LIN {X 0,Y 559.92,Z 996.15,A -85,B 0,C 180,E1 26542.512,E2 26542.512} C_VEL
LIN {X 0,Y 559.973,Z 989.657,A -85,B 0,C 180,E1 26540.271,E2 26540.271} C_VEL
LIN {X 0,Y 560.061,Z 982.262,A -85,B 0,C 180,E1 26538.26,E2 26538.26} C_VEL
LIN {X 0,Y 560.202,Z 972.761,A -85,B 0,C 180,E1 26536.152,E2 26536.152} C_VEL
LIN {X 0,Y 560.424,Z 961.483,A -85,B 0,C 180,E1 26534.055,E2 26534.055} C_VEL
LIN {X 0,Y 560.742,Z 948.646,A -85,B 0,C 180,E1 26532.035,E2 26532.035} C_VEL
LIN {X 0,Y 561.138,Z 934.193,A -85,B 0,C 180,E1 26530.106,E2 26530.106} C_VEL
LIN {X 0,Y 561.602,Z 918.797,A -85,B 0,C 180,E1 26528.333,E2 26528.333} C_VEL
LIN {X 0,Y 562.148,Z 901.727,A -85,B 0,C 180,E1 26526.635,E2 26526.635} C_VEL
LIN {X 0,Y 562.75,Z 883.794,A -85,B 0,C 180,E1 26525.1,E2 26525.1} C_VEL
LIN {X 0,Y 563.386,Z 864.761,A -85,B 0,C 180,E1 26523.721,E2 26523.721} C_VEL
LIN {X 0,Y 563.999,Z 844.815,A -85,B 0,C 180,E1 26522.499,E2 26522.499} C_VEL
LIN {X 0,Y 564.598,Z 825.21,A -85,B 0,C 180,E1 26521.497,E2 26521.497} C_VEL
LIN {X 0,Y 565.108,Z 804.841,A -85,B 0,C 180,E1 26520.656,E2 26520.656} C_VEL
LIN {X 0,Y 565.556,Z 782.74,A -85,B 0,C 180,E1 26519.949,E2 26519.949} C_VEL
LIN {X 0,Y 565.946,Z 761.19,A -85,B 0,C 180,E1 26519.454,E2 26519.454} C_VEL
LIN {X 0,Y 567.275,Z 543.866,A -85,B 0,C 180,E1 26516.321,E2 26516.321} C_VEL
LIN {X 0,Y 567.582,Z 462.459,A -85,B 0,C 180,E1 26515.12,E2 26515.12} C_VEL
LIN {X 0,Y 566.314,Z 454.968,A -85,B 0,C 180,E1 26514.909,E2 26514.909} C_VEL
LIN {X 0,Y 567.237,Z 411.986,A -85,B 0,C 180,E1 26512.196,E2 26512.196} C_VEL
LIN {X 0,Y 560.35,Z 396.389,A -85,B 0,C 180,E1 26510.568,E2 26510.568} C_VEL
LIN {X 0,Y 560.276,Z 395.939,A -85,B 0,C 180,E1 26510.278,E2 26510.278} C_VEL
LIN {X 0,Y 560.249,Z 395.947,A -85,B 0,C 180,E1 26507.025,E2 26507.025} C_VEL
LIN {X 0,Y 560.265,Z 395.941,A -85,B 0,C 180,E1 26503.681,E2 26503.681} C_VEL
LIN {X 0,Y 560.282,Z 395.942,A -85,B 0,C 180,E1 26500.364,E2 26500.364} C_VEL
LIN {X 0,Y 560.232,Z 395.947,A -85,B 0,C 180,E1 26497.088,E2 26497.088} C_VEL
LIN {X 0,Y 560.281,Z 395.945,A -85,B 0,C 180,E1 26493.833,E2 26493.833} C_VEL
LIN {X 0,Y 560.225,Z 395.947,A -85,B 0,C 180,E1 26490.663,E2 26490.663} C_VEL
LIN {X 0,Y 560.25,Z 395.947,A -85,B 0,C 180,E1 26487.415,E2 26487.415} C_VEL
LIN {X 0,Y 560.221,Z 395.947,A -85,B 0,C 180,E1 26484.348,E2 26484.348} C_VEL
LIN {X 0,Y 560.218,Z 395.947,A -85,B 0,C 180,E1 26481.022,E2 26481.022} C_VEL
LIN {X 0,Y 560.23,Z 395.948,A -85,B 0,C 180,E1 26477.975,E2 26477.975} C_VEL
LIN {X 0,Y 560.197,Z 395.947,A -85,B 0,C 180,E1 26474.681,E2 26474.681} C_VEL
LIN {X 0,Y 560.264,Z 395.947,A -85,B 0,C 180,E1 26471.529,E2 26471.529} C_VEL
LIN {X 0,Y 560.202,Z 395.946,A -85,B 0,C 180,E1 26468.312,E2 26468.312} C_VEL
LIN {X 0,Y 560.271,Z 395.946,A -85,B 0,C 180,E1 26465.119,E2 26465.119} C_VEL
LIN {X 0,Y 560.22,Z 395.946,A -85,B 0,C 180,E1 26461.943,E2 26461.943} C_VEL
LIN {X 0,Y 560.239,Z 395.945,A -85,B 0,C 180,E1 26458.568,E2 26458.568} C_VEL
LIN {X 0,Y 560.261,Z 395.946,A -85,B 0,C 180,E1 26455.393,E2 26455.393} C_VEL
LIN {X 0,Y 560.232,Z 395.946,A -85,B 0,C 180,E1 26452.076,E2 26452.076} C_VEL
LIN {X 0,Y 560.282,Z 395.944,A -85,B 0,C 180,E1 26448.887,E2 26448.887} C_VEL
LIN {X 0,Y 560.242,Z 395.946,A -85,B 0,C 180,E1 26445.636,E2 26445.636} C_VEL
LIN {X 0,Y 560.276,Z 395.941,A -85,B 0,C 180,E1 26442.339,E2 26442.339} C_VEL
LIN {X 0,Y 560.281,Z 395.941,A -85,B 0,C 180,E1 26438.949,E2 26438.949} C_VEL
LIN {X 0,Y 560.282,Z 395.941,A -85,B 0,C 180,E1 26436.242,E2 26436.242} C_VEL
LIN {X 0,Y 559.287,Z 396.064,A -85,B 0,C 180,E1 26435.455,E2 26435.455} C_VEL
LIN {X 0,Y 552.871,Z 396.865,A -85,B 0,C 180,E1 26433.243,E2 26433.243} C_VEL
LIN {X 0,Y 552.334,Z 396.924,A -85,B 0,C 180,E1 26432.667,E2 26432.667} C_VEL
LIN {X 0,Y 552.397,Z 397.316,A -85,B 0,C 180,E1 26432.24,E2 26432.24} C_VEL
LIN {X 0,Y 557.962,Z 412.47,A -85,B 0,C 180,E1 26430.505,E2 26430.505} C_VEL
LIN {X 0,Y 556.968,Z 452.354,A -85,B 0,C 180,E1 26427.431,E2 26427.431} C_VEL
LIN {X 0,Y 558.756,Z 463.241,A -85,B 0,C 180,E1 26427.151,E2 26427.151} C_VEL
LIN {X 0,Y 557.243,Z 713.555,A -85,B 0,C 180,E1 26423.618,E2 26423.618} C_VEL
LIN {X 0,Y 556.883,Z 733.935,A -85,B 0,C 180,E1 26423.144,E2 26423.144} C_VEL
LIN {X 0,Y 556.454,Z 753.084,A -85,B 0,C 180,E1 26422.519,E2 26422.519} C_VEL
LIN {X 0,Y 555.948,Z 772.8,A -85,B 0,C 180,E1 26421.682,E2 26421.682} C_VEL
LIN {X 0,Y 555.374,Z 791.75,A -85,B 0,C 180,E1 26420.675,E2 26420.675} C_VEL
LIN {X 0,Y 554.778,Z 810.212,A -85,B 0,C 180,E1 26419.478,E2 26419.478} C_VEL
LIN {X 0,Y 554.188,Z 827.589,A -85,B 0,C 180,E1 26418.121,E2 26418.121} C_VEL
LIN {X 0,Y 553.652,Z 843.71,A -85,B 0,C 180,E1 26416.633,E2 26416.633} C_VEL
LIN {X 0,Y 553.171,Z 858.492,A -85,B 0,C 180,E1 26415.03,E2 26415.03} C_VEL
LIN {X 0,Y 552.755,Z 872.818,A -85,B 0,C 180,E1 26413.199,E2 26413.199} C_VEL
LIN {X 0,Y 552.434,Z 885.237,A -85,B 0,C 180,E1 26411.313,E2 26411.313} C_VEL
LIN {X 0,Y 552.217,Z 895.965,A -85,B 0,C 180,E1 26409.363,E2 26409.363} C_VEL
LIN {X 0,Y 552.063,Z 905.093,A -85,B 0,C 180,E1 26407.349,E2 26407.349} C_VEL
LIN {X 0,Y 551.978,Z 912.761,A -85,B 0,C 180,E1 26405.219,E2 26405.219} C_VEL
LIN {X 0,Y 551.935,Z 918.327,A -85,B 0,C 180,E1 26403.164,E2 26403.164} C_VEL
LIN {X 0,Y 551.919,Z 922.392,A -85,B 0,C 180,E1 26401.03,E2 26401.03} C_VEL
LIN {X 0,Y 551.912,Z 924.818,A -85,B 0,C 180,E1 26398.806,E2 26398.806} C_VEL
LIN {X 0,Y 551.907,Z 925.449,A -85,B 0,C 180,E1 26396.695,E2 26396.695} C_VEL
LIN {X 0,Y 551.911,Z 924.457,A -85,B 0,C 180,E1 26394.571,E2 26394.571} C_VEL
LIN {X 0,Y 551.92,Z 921.593,A -85,B 0,C 180,E1 26392.358,E2 26392.358} C_VEL
LIN {X 0,Y 551.941,Z 917.367,A -85,B 0,C 180,E1 26390.351,E2 26390.351} C_VEL
LIN {X 0,Y 551.986,Z 911.309,A -85,B 0,C 180,E1 26388.259,E2 26388.259} C_VEL
LIN {X 0,Y 552.079,Z 903.952,A -85,B 0,C 180,E1 26386.285,E2 26386.285} C_VEL
LIN {X 0,Y 552.246,Z 894.517,A -85,B 0,C 180,E1 26384.252,E2 26384.252} C_VEL
LIN {X 0,Y 552.488,Z 883.101,A -85,B 0,C 180,E1 26382.241,E2 26382.241} C_VEL
LIN {X 0,Y 552.812,Z 870.701,A -85,B 0,C 180,E1 26380.418,E2 26380.418} C_VEL
LIN {X 0,Y 553.208,Z 857.202,A -85,B 0,C 180,E1 26378.73,E2 26378.73} C_VEL
LIN {X 0,Y 553.725,Z 841.406,A -85,B 0,C 180,E1 26377.051,E2 26377.051} C_VEL
LIN {X 0,Y 554.291,Z 824.528,A -85,B 0,C 180,E1 26375.536,E2 26375.536} C_VEL
LIN {X 0,Y 554.899,Z 806.565,A -85,B 0,C 180,E1 26374.183,E2 26374.183} C_VEL
LIN {X 0,Y 555.465,Z 788.406,A -85,B 0,C 180,E1 26373.042,E2 26373.042} C_VEL
LIN {X 0,Y 556.058,Z 769.286,A -85,B 0,C 180,E1 26372.059,E2 26372.059} C_VEL
LIN {X 0,Y 556.56,Z 749.527,A -85,B 0,C 180,E1 26371.259,E2 26371.259} C_VEL
LIN {X 0,Y 556.952,Z 729.557,A -85,B 0,C 180,E1 26370.649,E2 26370.649} C_VEL
LIN {X 0,Y 557.27,Z 708.606,A -85,B 0,C 180,E1 26370.21,E2 26370.21} C_VEL
LIN {X 0,Y 558.763,Z 462.012,A -85,B 0,C 180,E1 26366.741,E2 26366.741} C_VEL
LIN {X 0,Y 556.95,Z 451.832,A -85,B 0,C 180,E1 26366.447,E2 26366.447} C_VEL
LIN {X 0,Y 557.925,Z 412.19,A -85,B 0,C 180,E1 26363.384,E2 26363.384} C_VEL
LIN {X 0,Y 552.374,Z 397.163,A -85,B 0,C 180,E1 26361.672,E2 26361.672} C_VEL
LIN {X 0,Y 552.316,Z 396.929,A -85,B 0,C 180,E1 26358.3,E2 26358.3} C_VEL
LIN {X 0,Y 552.335,Z 396.934,A -85,B 0,C 180,E1 26354.996,E2 26354.996} C_VEL
LIN {X 0,Y 552.327,Z 396.925,A -85,B 0,C 180,E1 26351.638,E2 26351.638} C_VEL
LIN {X 0,Y 552.329,Z 396.919,A -85,B 0,C 180,E1 26348.215,E2 26348.215} C_VEL
LIN {X 0,Y 552.332,Z 396.929,A -85,B 0,C 180,E1 26344.822,E2 26344.822} C_VEL
LIN {X 0,Y 552.32,Z 396.932,A -85,B 0,C 180,E1 26341.567,E2 26341.567} C_VEL
LIN {X 0,Y 552.338,Z 396.931,A -85,B 0,C 180,E1 26338.211,E2 26338.211} C_VEL
LIN {X 0,Y 552.337,Z 396.923,A -85,B 0,C 180,E1 26334.853,E2 26334.853} C_VEL
LIN {X 0,Y 552.323,Z 396.929,A -85,B 0,C 180,E1 26331.448,E2 26331.448} C_VEL
LIN {X 0,Y 552.331,Z 396.933,A -85,B 0,C 180,E1 26328.087,E2 26328.087} C_VEL
LIN {X 0,Y 552.328,Z 396.929,A -85,B 0,C 180,E1 26324.765,E2 26324.765} C_VEL
LIN {X 0,Y 552.336,Z 396.932,A -85,B 0,C 180,E1 26321.3,E2 26321.3} C_VEL
LIN {X 0,Y 552.332,Z 396.929,A -85,B 0,C 180,E1 26317.988,E2 26317.988} C_VEL
LIN {X 0,Y 552.322,Z 396.932,A -85,B 0,C 180,E1 26314.641,E2 26314.641} C_VEL
LIN {X 0,Y 552.334,Z 396.93,A -85,B 0,C 180,E1 26311.301,E2 26311.301} C_VEL
LIN {X 0,Y 552.34,Z 396.927,A -85,B 0,C 180,E1 26307.843,E2 26307.843} C_VEL
LIN {X 0,Y 552.325,Z 396.932,A -85,B 0,C 180,E1 26304.415,E2 26304.415} C_VEL
LIN {X 0,Y 552.327,Z 396.931,A -85,B 0,C 180,E1 26301.115,E2 26301.115} C_VEL
LIN {X 0,Y 552.337,Z 396.928,A -85,B 0,C 180,E1 26297.706,E2 26297.706} C_VEL
LIN {X 0,Y 552.332,Z 396.931,A -85,B 0,C 180,E1 26294.253,E2 26294.253} C_VEL
LIN {X 0,Y 552.327,Z 396.931,A -85,B 0,C 180,E1 26290.958,E2 26290.958} C_VEL
LIN {X 0,Y 552.329,Z 396.928,A -85,B 0,C 180,E1 26287.594,E2 26287.594} C_VEL
LIN {X 0,Y 552.334,Z 396.934,A -85,B 0,C 180,E1 26284.257,E2 26284.257} C_VEL
LIN {X 0,Y 552.333,Z 396.928,A -85,B 0,C 180,E1 26280.83,E2 26280.83} C_VEL
LIN {X 0,Y 552.328,Z 396.931,A -85,B 0,C 180,E1 26277.51,E2 26277.51} C_VEL
LIN {X 0,Y 552.322,Z 396.933,A -85,B 0,C 180,E1 26274.182,E2 26274.182} C_VEL
LIN {X 0,Y 552.337,Z 396.928,A -85,B 0,C 180,E1 26270.834,E2 26270.834} C_VEL
LIN {X 0,Y 552.336,Z 396.933,A -85,B 0,C 180,E1 26267.348,E2 26267.348} C_VEL
LIN {X 0,Y 552.321,Z 396.93,A -85,B 0,C 180,E1 26264.001,E2 26264.001} C_VEL
LIN {X 0,Y 552.332,Z 396.93,A -85,B 0,C 180,E1 26260.654,E2 26260.654} C_VEL
LIN {X 0,Y 552.332,Z 396.934,A -85,B 0,C 180,E1 26257.32,E2 26257.32} C_VEL
LIN {X 0,Y 552.329,Z 396.929,A -85,B 0,C 180,E1 26253.883,E2 26253.883} C_VEL
LIN {X 0,Y 552.333,Z 396.934,A -85,B 0,C 180,E1 26250.545,E2 26250.545} C_VEL
LIN {X 0,Y 552.319,Z 396.931,A -85,B 0,C 180,E1 26247.23,E2 26247.23} C_VEL
LIN {X 0,Y 552.339,Z 396.93,A -85,B 0,C 180,E1 26243.834,E2 26243.834} C_VEL
LIN {X 0,Y 552.341,Z 396.934,A -85,B 0,C 180,E1 26240.417,E2 26240.417} C_VEL
LIN {X 0,Y 552.319,Z 396.932,A -85,B 0,C 180,E1 26237.104,E2 26237.104} C_VEL
LIN {X 0,Y 552.335,Z 396.933,A -85,B 0,C 180,E1 26233.751,E2 26233.751} C_VEL
LIN {X 0,Y 552.329,Z 396.929,A -85,B 0,C 180,E1 26230.349,E2 26230.349} C_VEL
LIN {X 0,Y 552.41,Z 397.394,A -85,B 0,C 180,E1 26230.038,E2 26230.038} C_VEL
LIN {X 0,Y 560.517,Z 415.82,A -85,B 0,C 180,E1 26228.081,E2 26228.081} C_VEL
LIN {X 0,Y 559.592,Z 455.684,A -85,B 0,C 180,E1 26225.558,E2 26225.558} C_VEL
LIN {X 0,Y 561.185,Z 466.213,A -85,B 0,C 180,E1 26225.279,E2 26225.279} C_VEL
LIN {X 0,Y 559.613,Z 686.518,A -85,B 0,C 180,E1 26222.062,E2 26222.062} C_VEL
LIN {X 0,Y 559.04,Z 762.278,A -85,B 0,C 180,E1 26220.946,E2 26220.946} C_VEL
LIN {X 0,Y 558.58,Z 783.721,A -85,B 0,C 180,E1 26220.437,E2 26220.437} C_VEL
LIN {X 0,Y 558.051,Z 805.52,A -85,B 0,C 180,E1 26219.724,E2 26219.724} C_VEL
LIN {X 0,Y 557.441,Z 826.358,A -85,B 0,C 180,E1 26218.85,E2 26218.85} C_VEL
LIN {X 0,Y 556.742,Z 845.724,A -85,B 0,C 180,E1 26217.837,E2 26217.837} C_VEL
LIN {X 0,Y 555.983,Z 866.308,A -85,B 0,C 180,E1 26216.546,E2 26216.546} C_VEL
LIN {X 0,Y 555.241,Z 885.093,A -85,B 0,C 180,E1 26215.151,E2 26215.151} C_VEL
LIN {X 0,Y 554.548,Z 902.884,A -85,B 0,C 180,E1 26213.597,E2 26213.597} C_VEL
LIN {X 0,Y 553.91,Z 919.519,A -85,B 0,C 180,E1 26211.904,E2 26211.904} C_VEL
LIN {X 0,Y 553.324,Z 935.858,A -85,B 0,C 180,E1 26209.971,E2 26209.971} C_VEL
LIN {X 0,Y 552.863,Z 950.032,A -85,B 0,C 180,E1 26208.016,E2 26208.016} C_VEL
LIN {X 0,Y 552.505,Z 962.724,A -85,B 0,C 180,E1 26205.968,E2 26205.968} C_VEL
LIN {X 0,Y 552.256,Z 973.324,A -85,B 0,C 180,E1 26203.935,E2 26203.935} C_VEL
LIN {X 0,Y 552.08,Z 983.061,A -85,B 0,C 180,E1 26201.705,E2 26201.705} C_VEL
LIN {X 0,Y 551.98,Z 990.584,A -85,B 0,C 180,E1 26199.595,E2 26199.595} C_VEL
LIN {X 0,Y 551.925,Z 996.394,A -85,B 0,C 180,E1 26197.497,E2 26197.497} C_VEL
LIN {X 0,Y 551.905,Z 1000.982,A -85,B 0,C 180,E1 26195.303,E2 26195.303} C_VEL
LIN {X 0,Y 551.907,Z 1003.783,A -85,B 0,C 180,E1 26193.222,E2 26193.222} C_VEL
LIN {X 0,Y 551.903,Z 1005.306,A -85,B 0,C 180,E1 26190.936,E2 26190.936} C_VEL
LIN {X 0,Y 551.909,Z 1005.238,A -85,B 0,C 180,E1 26188.757,E2 26188.757} C_VEL
LIN {X 0,Y 551.914,Z 1003.545,A -85,B 0,C 180,E1 26186.559,E2 26186.559} C_VEL
LIN {X 0,Y 551.925,Z 1000.225,A -85,B 0,C 180,E1 26184.284,E2 26184.284} C_VEL
LIN {X 0,Y 551.946,Z 995.642,A -85,B 0,C 180,E1 26182.194,E2 26182.194} C_VEL
LIN {X 0,Y 552.003,Z 989.184,A -85,B 0,C 180,E1 26179.989,E2 26179.989} C_VEL
LIN {X 0,Y 552.117,Z 981.441,A -85,B 0,C 180,E1 26177.876,E2 26177.876} C_VEL
LIN {X 0,Y 552.296,Z 971.788,A -85,B 0,C 180,E1 26175.749,E2 26175.749} C_VEL
LIN {X 0,Y 552.579,Z 960.21,A -85,B 0,C 180,E1 26173.607,E2 26173.607} C_VEL
LIN {X 0,Y 552.936,Z 947.895,A -85,B 0,C 180,E1 26171.664,E2 26171.664} C_VEL
LIN {X 0,Y 553.409,Z 933.343,A -85,B 0,C 180,E1 26169.706,E2 26169.706} C_VEL
LIN {X 0,Y 553.971,Z 917.688,A -85,B 0,C 180,E1 26167.897,E2 26167.897} C_VEL
LIN {X 0,Y 554.661,Z 899.917,A -85,B 0,C 180,E1 26166.131,E2 26166.131} C_VEL
LIN {X 0,Y 555.379,Z 881.775,A -85,B 0,C 180,E1 26164.588,E2 26164.588} C_VEL
LIN {X 0,Y 556.106,Z 863.135,A -85,B 0,C 180,E1 26163.235,E2 26163.235} C_VEL
LIN {X 0,Y 556.812,Z 843.817,A -85,B 0,C 180,E1 26162.055,E2 26162.055} C_VEL
LIN {X 0,Y 557.492,Z 823.942,A -85,B 0,C 180,E1 26161.041,E2 26161.041} C_VEL
LIN {X 0,Y 558.103,Z 804.099,A -85,B 0,C 180,E1 26160.222,E2 26160.222} C_VEL
LIN {X 0,Y 558.603,Z 782.221,A -85,B 0,C 180,E1 26159.521,E2 26159.521} C_VEL
LIN {X 0,Y 559.058,Z 760.334,A -85,B 0,C 180,E1 26159.021,E2 26159.021} C_VEL
LIN {X 0,Y 560.682,Z 534.694,A -85,B 0,C 180,E1 26155.731,E2 26155.731} C_VEL
LIN {X 0,Y 561.012,Z 463.917,A -85,B 0,C 180,E1 26154.674,E2 26154.674} C_VEL
LIN {X 0,Y 559.495,Z 454.665,A -85,B 0,C 180,E1 26154.401,E2 26154.401} C_VEL
LIN {X 0,Y 560.46,Z 415.329,A -85,B 0,C 180,E1 26151.882,E2 26151.882} C_VEL
LIN {X 0,Y 552.396,Z 397.288,A -85,B 0,C 180,E1 26149.945,E2 26149.945} C_VEL
LIN {X 0,Y 552.312,Z 396.928,A -85,B 0,C 180,E1 26149.175,E2 26149.175} C_VEL
LIN {X 0,Y 552.333,Z 396.928,A -85,B 0,C 180,E1 26145.795,E2 26145.795} C_VEL
LIN {X 0,Y 552.338,Z 396.923,A -85,B 0,C 180,E1 26142.395,E2 26142.395} C_VEL
LIN {X 0,Y 552.298,Z 396.936,A -85,B 0,C 180,E1 26139.184,E2 26139.184} C_VEL
LIN {X 0,Y 552.344,Z 396.934,A -85,B 0,C 180,E1 26135.909,E2 26135.909} C_VEL
LIN {X 0,Y 552.293,Z 396.935,A -85,B 0,C 180,E1 26132.649,E2 26132.649} C_VEL
LIN {X 0,Y 552.296,Z 396.937,A -85,B 0,C 180,E1 26129.246,E2 26129.246} C_VEL
LIN {X 0,Y 552.31,Z 396.932,A -85,B 0,C 180,E1 26126.123,E2 26126.123} C_VEL
LIN {X 0,Y 552.274,Z 396.938,A -85,B 0,C 180,E1 26122.862,E2 26122.862} C_VEL
LIN {X 0,Y 552.332,Z 396.935,A -85,B 0,C 180,E1 26119.676,E2 26119.676} C_VEL
LIN {X 0,Y 552.258,Z 396.939,A -85,B 0,C 180,E1 26116.514,E2 26116.514} C_VEL
LIN {X 0,Y 552.316,Z 396.938,A -85,B 0,C 180,E1 26113.291,E2 26113.291} C_VEL
LIN {X 0,Y 552.263,Z 396.938,A -85,B 0,C 180,E1 26110.22,E2 26110.22} C_VEL
LIN {X 0,Y 552.306,Z 396.936,A -85,B 0,C 180,E1 26106.966,E2 26106.966} C_VEL
LIN {X 0,Y 552.286,Z 396.937,A -85,B 0,C 180,E1 26103.841,E2 26103.841} C_VEL
LIN {X 0,Y 552.286,Z 396.935,A -85,B 0,C 180,E1 26100.415,E2 26100.415} C_VEL
LIN {X 0,Y 552.341,Z 396.935,A -85,B 0,C 180,E1 26097.198,E2 26097.198} C_VEL
LIN {X 0,Y 552.289,Z 396.935,A -85,B 0,C 180,E1 26093.972,E2 26093.972} C_VEL
LIN {X 0,Y 552.34,Z 396.932,A -85,B 0,C 180,E1 26090.728,E2 26090.728} C_VEL
LIN {X 0,Y 552.313,Z 396.937,A -85,B 0,C 180,E1 26087.453,E2 26087.453} C_VEL
LIN {X 0,Y 552.311,Z 396.932,A -85,B 0,C 180,E1 26084.028,E2 26084.028} C_VEL
LIN {X 0,Y 552.34,Z 396.934,A -85,B 0,C 180,E1 26080.764,E2 26080.764} C_VEL
LIN {X 0,Y 552.315,Z 396.929,A -85,B 0,C 180,E1 26077.431,E2 26077.431} C_VEL
LIN {X 0,Y 552.336,Z 396.935,A -85,B 0,C 180,E1 26074.018,E2 26074.018} C_VEL
LIN {X 0,Y 552.334,Z 396.924,A -85,B 0,C 180,E1 26072.667,E2 26072.667} C_VEL
LIN {X 0,Y 552.297,Z 397.934,A -85,B 0,C 180,E1 26072.317,E2 26072.317} C_VEL
LIN {X 0,Y 552.136,Z 402.018,A -85,B 0,C 180,E1 26071.841,E2 26071.841} C_VEL
LIN {X 0,Y 550.706,Z 423.331,A -85,B 0,C 180,E1 26070.151,E2 26070.151} C_VEL
LIN {X 0,Y 549.819,Z 452.552,A -85,B 0,C 180,E1 26067.865,E2 26067.865} C_VEL
LIN {X 0,Y 551.832,Z 464.588,A -85,B 0,C 180,E1 26067.551,E2 26067.551} C_VEL
LIN {X 0,Y 550.09,Z 713.472,A -85,B 0,C 180,E1 26063.995,E2 26063.995} C_VEL
LIN {X 0,Y 549.677,Z 733.913,A -85,B 0,C 180,E1 26063.515,E2 26063.515} C_VEL
LIN {X 0,Y 549.192,Z 753.177,A -85,B 0,C 180,E1 26062.879,E2 26062.879} C_VEL
LIN {X 0,Y 548.586,Z 773.344,A -85,B 0,C 180,E1 26062.008,E2 26062.008} C_VEL
LIN {X 0,Y 547.917,Z 792.321,A -85,B 0,C 180,E1 26060.981,E2 26060.981} C_VEL
LIN {X 0,Y 547.231,Z 810.861,A -85,B 0,C 180,E1 26059.756,E2 26059.756} C_VEL
LIN {X 0,Y 546.528,Z 828.961,A -85,B 0,C 180,E1 26058.315,E2 26058.315} C_VEL
LIN {X 0,Y 545.887,Z 845.633,A -85,B 0,C 180,E1 26056.73,E2 26056.73} C_VEL
LIN {X 0,Y 545.325,Z 860.61,A -85,B 0,C 180,E1 26055.046,E2 26055.046} C_VEL
LIN {X 0,Y 544.86,Z 874.255,A -85,B 0,C 180,E1 26053.237,E2 26053.237} C_VEL
LIN {X 0,Y 544.498,Z 886.454,A -85,B 0,C 180,E1 26051.319,E2 26051.319} C_VEL
LIN {X 0,Y 544.24,Z 897.278,A -85,B 0,C 180,E1 26049.275,E2 26049.275} C_VEL
LIN {X 0,Y 544.067,Z 906.256,A -85,B 0,C 180,E1 26047.197,E2 26047.197} C_VEL
LIN {X 0,Y 543.981,Z 913.418,A -85,B 0,C 180,E1 26045.117,E2 26045.117} C_VEL
LIN {X 0,Y 543.937,Z 919.031,A -85,B 0,C 180,E1 26042.96,E2 26042.96} C_VEL
LIN {X 0,Y 543.922,Z 922.75,A -85,B 0,C 180,E1 26040.851,E2 26040.851} C_VEL
LIN {X 0,Y 543.907,Z 924.922,A -85,B 0,C 180,E1 26038.668,E2 26038.668} C_VEL
LIN {X 0,Y 543.903,Z 925.39,A -85,B 0,C 180,E1 26036.412,E2 26036.412} C_VEL
LIN {X 0,Y 543.912,Z 924.151,A -85,B 0,C 180,E1 26034.246,E2 26034.246} C_VEL
LIN {X 0,Y 543.923,Z 921.293,A -85,B 0,C 180,E1 26032.108,E2 26032.108} C_VEL
LIN {X 0,Y 543.943,Z 916.735,A -85,B 0,C 180,E1 26029.99,E2 26029.99} C_VEL
LIN {X 0,Y 543.999,Z 910.818,A -85,B 0,C 180,E1 26027.983,E2 26027.983} C_VEL
LIN {X 0,Y 544.12,Z 902.924,A -85,B 0,C 180,E1 26025.888,E2 26025.888} C_VEL
LIN {X 0,Y 544.322,Z 893.767,A -85,B 0,C 180,E1 26023.921,E2 26023.921} C_VEL
LIN {X 0,Y 544.625,Z 882.329,A -85,B 0,C 180,E1 26021.896,E2 26021.896} C_VEL
LIN {X 0,Y 545.005,Z 869.718,A -85,B 0,C 180,E1 26020.034,E2 26020.034} C_VEL
LIN {X 0,Y 545.478,Z 856.038,A -85,B 0,C 180,E1 26018.324,E2 26018.324} C_VEL
LIN {X 0,Y 546.039,Z 841.098,A -85,B 0,C 180,E1 26016.728,E2 26016.728} C_VEL
LIN {X 0,Y 546.707,Z 824.144,A -85,B 0,C 180,E1 26015.191,E2 26015.191} C_VEL
LIN {X 0,Y 547.416,Z 806.094,A -85,B 0,C 180,E1 26013.82,E2 26013.82} C_VEL
LIN {X 0,Y 548.082,Z 787.805,A -85,B 0,C 180,E1 26012.664,E2 26012.664} C_VEL
LIN {X 0,Y 548.747,Z 768.515,A -85,B 0,C 180,E1 26011.668,E2 26011.668} C_VEL
LIN {X 0,Y 549.339,Z 748.562,A -85,B 0,C 180,E1 26010.858,E2 26010.858} C_VEL
LIN {X 0,Y 549.8,Z 728.444,A -85,B 0,C 180,E1 26010.248,E2 26010.248} C_VEL
LIN {X 0,Y 550.127,Z 707.886,A -85,B 0,C 180,E1 26009.822,E2 26009.822} C_VEL
LIN {X 0,Y 551.842,Z 463.422,A -85,B 0,C 180,E1 26006.343,E2 26006.343} C_VEL
LIN {X 0,Y 549.793,Z 452.315,A -85,B 0,C 180,E1 26006.035,E2 26006.035} C_VEL
LIN {X 0,Y 550.947,Z 415.541,A -85,B 0,C 180,E1 26003.142,E2 26003.142} C_VEL
LIN {X 0,Y 545.067,Z 400.264,A -85,B 0,C 180,E1 26001.392,E2 26001.392} C_VEL
LIN {X 0,Y 544.423,Z 398.102,A -85,B 0,C 180,E1 26001.097,E2 26001.097} C_VEL
LIN {X 0,Y 544.395,Z 397.906,A -85,B 0,C 180,E1 25997.697,E2 25997.697} C_VEL
LIN {X 0,Y 544.383,Z 397.92,A -85,B 0,C 180,E1 25994.244,E2 25994.244} C_VEL
LIN {X 0,Y 544.394,Z 397.916,A -85,B 0,C 180,E1 25990.916,E2 25990.916} C_VEL
LIN {X 0,Y 544.384,Z 397.9,A -85,B 0,C 180,E1 25987.539,E2 25987.539} C_VEL
LIN {X 0,Y 544.393,Z 397.925,A -85,B 0,C 180,E1 25984.078,E2 25984.078} C_VEL
LIN {X 0,Y 544.395,Z 397.92,A -85,B 0,C 180,E1 25980.74,E2 25980.74} C_VEL
LIN {X 0,Y 544.381,Z 397.922,A -85,B 0,C 180,E1 25977.441,E2 25977.441} C_VEL
LIN {X 0,Y 544.401,Z 397.92,A -85,B 0,C 180,E1 25974.003,E2 25974.003} C_VEL
LIN {X 0,Y 544.4,Z 397.911,A -85,B 0,C 180,E1 25970.544,E2 25970.544} C_VEL
LIN {X 0,Y 544.383,Z 397.915,A -85,B 0,C 180,E1 25967.188,E2 25967.188} C_VEL
LIN {X 0,Y 544.394,Z 397.923,A -85,B 0,C 180,E1 25963.822,E2 25963.822} C_VEL
LIN {X 0,Y 544.405,Z 397.914,A -85,B 0,C 180,E1 25960.341,E2 25960.341} C_VEL
LIN {X 0,Y 544.385,Z 397.917,A -85,B 0,C 180,E1 25956.913,E2 25956.913} C_VEL
LIN {X 0,Y 544.39,Z 397.923,A -85,B 0,C 180,E1 25953.503,E2 25953.503} C_VEL
LIN {X 0,Y 544.402,Z 397.914,A -85,B 0,C 180,E1 25950.093,E2 25950.093} C_VEL
LIN {X 0,Y 544.389,Z 397.915,A -85,B 0,C 180,E1 25946.625,E2 25946.625} C_VEL
LIN {X 0,Y 544.389,Z 397.92,A -85,B 0,C 180,E1 25943.259,E2 25943.259} C_VEL
LIN {X 0,Y 544.393,Z 397.911,A -85,B 0,C 180,E1 25939.864,E2 25939.864} C_VEL
LIN {X 0,Y 544.398,Z 397.922,A -85,B 0,C 180,E1 25936.43,E2 25936.43} C_VEL
LIN {X 0,Y 544.388,Z 397.916,A -85,B 0,C 180,E1 25933.057,E2 25933.057} C_VEL
LIN {X 0,Y 544.388,Z 397.914,A -85,B 0,C 180,E1 25929.728,E2 25929.728} C_VEL
LIN {X 0,Y 544.397,Z 397.923,A -85,B 0,C 180,E1 25926.327,E2 25926.327} C_VEL
LIN {X 0,Y 544.39,Z 397.91,A -85,B 0,C 180,E1 25922.843,E2 25922.843} C_VEL
LIN {X 0,Y 544.389,Z 397.918,A -85,B 0,C 180,E1 25919.474,E2 25919.474} C_VEL
LIN {X 0,Y 544.389,Z 397.92,A -85,B 0,C 180,E1 25916.104,E2 25916.104} C_VEL
LIN {X 0,Y 544.396,Z 397.909,A -85,B 0,C 180,E1 25912.614,E2 25912.614} C_VEL
LIN {X 0,Y 544.392,Z 397.919,A -85,B 0,C 180,E1 25909.203,E2 25909.203} C_VEL
LIN {X 0,Y 544.385,Z 397.921,A -85,B 0,C 180,E1 25905.861,E2 25905.861} C_VEL
LIN {X 0,Y 544.399,Z 397.915,A -85,B 0,C 180,E1 25902.47,E2 25902.47} C_VEL
LIN {X 0,Y 544.398,Z 397.919,A -85,B 0,C 180,E1 25899.014,E2 25899.014} C_VEL
LIN {X 0,Y 544.38,Z 397.921,A -85,B 0,C 180,E1 25895.645,E2 25895.645} C_VEL
LIN {X 0,Y 544.398,Z 397.916,A -85,B 0,C 180,E1 25892.284,E2 25892.284} C_VEL
LIN {X 0,Y 544.402,Z 397.922,A -85,B 0,C 180,E1 25888.807,E2 25888.807} C_VEL
LIN {X 0,Y 544.381,Z 397.921,A -85,B 0,C 180,E1 25885.371,E2 25885.371} C_VEL
LIN {X 0,Y 544.396,Z 397.919,A -85,B 0,C 180,E1 25881.993,E2 25881.993} C_VEL
LIN {X 0,Y 544.395,Z 397.923,A -85,B 0,C 180,E1 25878.61,E2 25878.61} C_VEL
LIN {X 0,Y 544.381,Z 397.908,A -85,B 0,C 180,E1 25875.148,E2 25875.148} C_VEL
LIN {X 0,Y 544.391,Z 397.897,A -85,B 0,C 180,E1 25871.815,E2 25871.815} C_VEL
LIN {X 0,Y 544.413,Z 398.164,A -85,B 0,C 180,E1 25870.668,E2 25870.668} C_VEL
LIN {X 0,Y 545.523,Z 401.136,A -85,B 0,C 180,E1 25870.317,E2 25870.317} C_VEL
LIN {X 0,Y 553.767,Z 419.076,A -85,B 0,C 180,E1 25868.408,E2 25868.408} C_VEL
LIN {X 0,Y 552.808,Z 455.62,A -85,B 0,C 180,E1 25866.063,E2 25866.063} C_VEL
LIN {X 0,Y 554.641,Z 467.677,A -85,B 0,C 180,E1 25865.735,E2 25865.735} C_VEL
LIN {X 0,Y 552.823,Z 687.917,A -85,B 0,C 180,E1 25862.483,E2 25862.483} C_VEL
LIN {X 0,Y 552.175,Z 762.278,A -85,B 0,C 180,E1 25861.374,E2 25861.374} C_VEL
LIN {X 0,Y 551.643,Z 783.852,A -85,B 0,C 180,E1 25860.858,E2 25860.858} C_VEL
LIN {X 0,Y 551.021,Z 806.182,A -85,B 0,C 180,E1 25860.116,E2 25860.116} C_VEL
LIN {X 0,Y 550.334,Z 826.358,A -85,B 0,C 180,E1 25859.258,E2 25859.258} C_VEL
LIN {X 0,Y 549.541,Z 845.727,A -85,B 0,C 180,E1 25858.234,E2 25858.234} C_VEL
LIN {X 0,Y 548.658,Z 866.305,A -85,B 0,C 180,E1 25856.929,E2 25856.929} C_VEL
LIN {X 0,Y 547.805,Z 885.09,A -85,B 0,C 180,E1 25855.517,E2 25855.517} C_VEL
LIN {X 0,Y 547.005,Z 902.886,A -85,B 0,C 180,E1 25853.942,E2 25853.942} C_VEL
LIN {X 0,Y 546.266,Z 919.164,A -85,B 0,C 180,E1 25852.266,E2 25852.266} C_VEL
LIN {X 0,Y 545.603,Z 935.008,A -85,B 0,C 180,E1 25850.378,E2 25850.378} C_VEL
LIN {X 0,Y 545.097,Z 948.63,A -85,B 0,C 180,E1 25848.501,E2 25848.501} C_VEL
LIN {X 0,Y 544.663,Z 961.453,A -85,B 0,C 180,E1 25846.423,E2 25846.423} C_VEL
LIN {X 0,Y 544.341,Z 972.806,A -85,B 0,C 180,E1 25844.251,E2 25844.251} C_VEL
LIN {X 0,Y 544.136,Z 982.247,A -85,B 0,C 180,E1 25842.094,E2 25842.094} C_VEL
LIN {X 0,Y 544.009,Z 989.877,A -85,B 0,C 180,E1 25839.951,E2 25839.951} C_VEL
LIN {X 0,Y 543.942,Z 996.14,A -85,B 0,C 180,E1 25837.714,E2 25837.714} C_VEL
LIN {X 0,Y 543.916,Z 1000.821,A -85,B 0,C 180,E1 25835.487,E2 25835.487} C_VEL
LIN {X 0,Y 543.909,Z 1003.783,A -85,B 0,C 180,E1 25833.269,E2 25833.269} C_VEL
LIN {X 0,Y 543.905,Z 1005.306,A -85,B 0,C 180,E1 25830.95,E2 25830.95} C_VEL
LIN {X 0,Y 543.908,Z 1005.238,A -85,B 0,C 180,E1 25828.738,E2 25828.738} C_VEL
LIN {X 0,Y 543.913,Z 1003.562,A -85,B 0,C 180,E1 25826.524,E2 25826.524} C_VEL
LIN {X 0,Y 543.925,Z 1000.431,A -85,B 0,C 180,E1 25824.306,E2 25824.306} C_VEL
LIN {X 0,Y 543.95,Z 995.896,A -85,B 0,C 180,E1 25822.185,E2 25822.185} C_VEL
LIN {X 0,Y 544.03,Z 989.185,A -85,B 0,C 180,E1 25819.84,E2 25819.84} C_VEL
LIN {X 0,Y 544.161,Z 981.441,A -85,B 0,C 180,E1 25817.696,E2 25817.696} C_VEL
LIN {X 0,Y 544.375,Z 971.789,A -85,B 0,C 180,E1 25815.538,E2 25815.538} C_VEL
LIN {X 0,Y 544.705,Z 960.21,A -85,B 0,C 180,E1 25813.363,E2 25813.363} C_VEL
LIN {X 0,Y 545.123,Z 947.894,A -85,B 0,C 180,E1 25811.392,E2 25811.392} C_VEL
LIN {X 0,Y 545.672,Z 933.344,A -85,B 0,C 180,E1 25809.405,E2 25809.405} C_VEL
LIN {X 0,Y 546.303,Z 918.194,A -85,B 0,C 180,E1 25807.627,E2 25807.627} C_VEL
LIN {X 0,Y 547.106,Z 900.522,A -85,B 0,C 180,E1 25805.838,E2 25805.838} C_VEL
LIN {X 0,Y 547.914,Z 883.073,A -85,B 0,C 180,E1 25804.32,E2 25804.32} C_VEL
LIN {X 0,Y 548.728,Z 864.64,A -85,B 0,C 180,E1 25802.954,E2 25802.954} C_VEL
LIN {X 0,Y 549.583,Z 844.708,A -85,B 0,C 180,E1 25801.707,E2 25801.707} C_VEL
LIN {X 0,Y 550.381,Z 824.65,A -85,B 0,C 180,E1 25800.663,E2 25800.663} C_VEL
LIN {X 0,Y 551.074,Z 804.836,A -85,B 0,C 180,E1 25799.833,E2 25799.833} C_VEL
LIN {X 0,Y 551.669,Z 782.611,A -85,B 0,C 180,E1 25799.108,E2 25799.108} C_VEL
LIN {X 0,Y 552.189,Z 760.869,A -85,B 0,C 180,E1 25798.602,E2 25798.602} C_VEL
LIN {X 0,Y 554.048,Z 537.366,A -85,B 0,C 180,E1 25795.304,E2 25795.304} C_VEL
LIN {X 0,Y 554.457,Z 465.295,A -85,B 0,C 180,E1 25794.214,E2 25794.214} C_VEL
LIN {X 0,Y 552.721,Z 454.694,A -85,B 0,C 180,E1 25793.899,E2 25793.899} C_VEL
LIN {X 0,Y 553.768,Z 419.073,A -85,B 0,C 180,E1 25791.592,E2 25791.592} C_VEL
LIN {X 0,Y 546.834,Z 404.135,A -85,B 0,C 180,E1 25790.006,E2 25790.006} C_VEL
LIN {X 0,Y 544.412,Z 398.202,A -85,B 0,C 180,E1 25789.355,E2 25789.355} C_VEL
LIN {X 0,Y 544.37,Z 397.926,A -85,B 0,C 180,E1 25787.126,E2 25787.126} C_VEL
LIN {X 0,Y 544.396,Z 397.918,A -85,B 0,C 180,E1 25783.802,E2 25783.802} C_VEL
LIN {X 0,Y 544.399,Z 397.921,A -85,B 0,C 180,E1 25780.415,E2 25780.415} C_VEL
LIN {X 0,Y 544.354,Z 397.925,A -85,B 0,C 180,E1 25777.046,E2 25777.046} C_VEL
LIN {X 0,Y 544.402,Z 397.923,A -85,B 0,C 180,E1 25773.813,E2 25773.813} C_VEL
LIN {X 0,Y 544.355,Z 397.924,A -85,B 0,C 180,E1 25770.528,E2 25770.528} C_VEL
LIN {X 0,Y 544.346,Z 397.923,A -85,B 0,C 180,E1 25767.099,E2 25767.099} C_VEL
LIN {X 0,Y 544.381,Z 397.924,A -85,B 0,C 180,E1 25763.948,E2 25763.948} C_VEL
LIN {X 0,Y 544.329,Z 397.925,A -85,B 0,C 180,E1 25760.763,E2 25760.763} C_VEL
LIN {X 0,Y 544.391,Z 397.923,A -85,B 0,C 180,E1 25757.53,E2 25757.53} C_VEL
LIN {X 0,Y 544.317,Z 397.925,A -85,B 0,C 180,E1 25754.358,E2 25754.358} C_VEL
LIN {X 0,Y 544.354,Z 397.927,A -85,B 0,C 180,E1 25751.012,E2 25751.012} C_VEL
LIN {X 0,Y 544.342,Z 397.923,A -85,B 0,C 180,E1 25747.918,E2 25747.918} C_VEL
LIN {X 0,Y 544.34,Z 397.925,A -85,B 0,C 180,E1 25744.53,E2 25744.53} C_VEL
LIN {X 0,Y 544.403,Z 397.923,A -85,B 0,C 180,E1 25741.263,E2 25741.263} C_VEL
LIN {X 0,Y 544.345,Z 397.925,A -85,B 0,C 180,E1 25738,E2 25738} C_VEL
LIN {X 0,Y 544.382,Z 397.921,A -85,B 0,C 180,E1 25734.625,E2 25734.625} C_VEL
LIN {X 0,Y 544.387,Z 397.926,A -85,B 0,C 180,E1 25731.338,E2 25731.338} C_VEL
LIN {X 0,Y 544.362,Z 397.923,A -85,B 0,C 180,E1 25728.021,E2 25728.021} C_VEL
LIN {X 0,Y 544.404,Z 397.921,A -85,B 0,C 180,E1 25724.773,E2 25724.773} C_VEL
LIN {X 0,Y 544.38,Z 397.926,A -85,B 0,C 180,E1 25721.381,E2 25721.381} C_VEL
LIN {X 0,Y 544.38,Z 397.913,A -85,B 0,C 180,E1 25717.881,E2 25717.881} C_VEL
LIN {X 0,Y 544.396,Z 397.918,A -85,B 0,C 180,E1 25714.546,E2 25714.546} C_VEL
LIN {X 0,Y 544.44,Z 398.198,A -85,B 0,C 180,E1 25712.83,E2 25712.83} C_VEL
LIN {X 0,Y 551.013,Z 415.543,A -85,B 0,C 180,E1 25710.782,E2 25710.782} C_VEL
LIN {X 0,Y 550.706,Z 423.331,A -85,B 0,C 180,E1 25710.151,E2 25710.151} C_VEL
LIN {X 0,Y 549.667,Z 427.669,A -85,B 0,C 180,E1 25709.867,E2 25709.867} C_VEL
LIN {X 0,Y 543.829,Z 439.733,A -85,B 0,C 180,E1 25709.295,E2 25709.295} C_VEL
LIN {X 0,Y 543.008,Z 443.458,A -85,B 0,C 180,E1 25709.044,E2 25709.044} C_VEL
LIN {X 0,Y 542.791,Z 452.86,A -85,B 0,C 180,E1 25708.324,E2 25708.324} C_VEL
LIN {X 0,Y 544.936,Z 465.984,A -85,B 0,C 180,E1 25707.959,E2 25707.959} C_VEL
LIN {X 0,Y 542.961,Z 713.427,A -85,B 0,C 180,E1 25704.38,E2 25704.38} C_VEL
LIN {X 0,Y 542.496,Z 733.915,A -85,B 0,C 180,E1 25703.895,E2 25703.895} C_VEL
LIN {X 0,Y 541.95,Z 753.328,A -85,B 0,C 180,E1 25703.245,E2 25703.245} C_VEL
LIN {X 0,Y 541.269,Z 773.177,A -85,B 0,C 180,E1 25702.379,E2 25702.379} C_VEL
LIN {X 0,Y 540.53,Z 791.732,A -85,B 0,C 180,E1 25701.369,E2 25701.369} C_VEL
LIN {X 0,Y 539.765,Z 810.232,A -85,B 0,C 180,E1 25700.139,E2 25700.139} C_VEL
LIN {X 0,Y 538.966,Z 828.16,A -85,B 0,C 180,E1 25698.7,E2 25698.7} C_VEL
LIN {X 0,Y 538.232,Z 844.586,A -85,B 0,C 180,E1 25697.131,E2 25697.131} C_VEL
LIN {X 0,Y 537.593,Z 859.267,A -85,B 0,C 180,E1 25695.478,E2 25695.478} C_VEL
LIN {X 0,Y 537.061,Z 872.865,A -85,B 0,C 180,E1 25693.681,E2 25693.681} C_VEL
LIN {X 0,Y 536.62,Z 885.547,A -85,B 0,C 180,E1 25691.692,E2 25691.692} C_VEL
LIN {X 0,Y 536.315,Z 896.577,A -85,B 0,C 180,E1 25689.608,E2 25689.608} C_VEL
LIN {X 0,Y 536.112,Z 905.448,A -85,B 0,C 180,E1 25687.567,E2 25687.567} C_VEL
LIN {X 0,Y 536,Z 912.984,A -85,B 0,C 180,E1 25685.394,E2 25685.394} C_VEL
LIN {X 0,Y 535.941,Z 918.54,A -85,B 0,C 180,E1 25683.26,E2 25683.26} C_VEL
LIN {X 0,Y 535.919,Z 922.485,A -85,B 0,C 180,E1 25681.09,E2 25681.09} C_VEL
LIN {X 0,Y 535.915,Z 924.797,A -85,B 0,C 180,E1 25678.892,E2 25678.892} C_VEL
LIN {X 0,Y 535.909,Z 925.455,A -85,B 0,C 180,E1 25676.717,E2 25676.717} C_VEL
LIN {X 0,Y 535.912,Z 924.522,A -85,B 0,C 180,E1 25674.582,E2 25674.582} C_VEL
LIN {X 0,Y 535.921,Z 921.812,A -85,B 0,C 180,E1 25672.368,E2 25672.368} C_VEL
LIN {X 0,Y 535.949,Z 917.447,A -85,B 0,C 180,E1 25670.187,E2 25670.187} C_VEL
LIN {X 0,Y 536.011,Z 911.14,A -85,B 0,C 180,E1 25667.947,E2 25667.947} C_VEL
LIN {X 0,Y 536.141,Z 903.714,A -85,B 0,C 180,E1 25665.908,E2 25665.908} C_VEL
LIN {X 0,Y 536.382,Z 894.167,A -85,B 0,C 180,E1 25663.801,E2 25663.801} C_VEL
LIN {X 0,Y 536.732,Z 882.596,A -85,B 0,C 180,E1 25661.713,E2 25661.713} C_VEL
LIN {X 0,Y 537.195,Z 869.496,A -85,B 0,C 180,E1 25659.749,E2 25659.749} C_VEL
LIN {X 0,Y 537.784,Z 854.872,A -85,B 0,C 180,E1 25657.905,E2 25657.905} C_VEL
LIN {X 0,Y 538.431,Z 839.712,A -85,B 0,C 180,E1 25656.288,E2 25656.288} C_VEL
LIN {X 0,Y 539.166,Z 823.13,A -85,B 0,C 180,E1 25654.784,E2 25654.784} C_VEL
LIN {X 0,Y 539.982,Z 804.85,A -85,B 0,C 180,E1 25653.395,E2 25653.395} C_VEL
LIN {X 0,Y 540.761,Z 786.251,A -85,B 0,C 180,E1 25652.223,E2 25652.223} C_VEL
LIN {X 0,Y 541.473,Z 767.722,A -85,B 0,C 180,E1 25651.267,E2 25651.267} C_VEL
LIN {X 0,Y 542.147,Z 747.386,A -85,B 0,C 180,E1 25650.44,E2 25650.44} C_VEL
LIN {X 0,Y 542.697,Z 726.764,A -85,B 0,C 180,E1 25649.823,E2 25649.823} C_VEL
LIN {X 0,Y 543.03,Z 706.253,A -85,B 0,C 180,E1 25649.409,E2 25649.409} C_VEL
LIN {X 0,Y 544.948,Z 464.839,A -85,B 0,C 180,E1 25645.934,E2 25645.934} C_VEL
LIN {X 0,Y 542.685,Z 452.145,A -85,B 0,C 180,E1 25645.56,E2 25645.56} C_VEL
LIN {X 0,Y 543.91,Z 418.664,A -85,B 0,C 180,E1 25642.87,E2 25642.87} C_VEL
LIN {X 0,Y 537.414,Z 401.808,A -85,B 0,C 180,E1 25640.899,E2 25640.899} C_VEL
LIN {X 0,Y 536.473,Z 399.104,A -85,B 0,C 180,E1 25640.531,E2 25640.531} C_VEL
LIN {X 0,Y 536.454,Z 398.89,A -85,B 0,C 180,E1 25637.184,E2 25637.184} C_VEL
LIN {X 0,Y 536.44,Z 398.905,A -85,B 0,C 180,E1 25633.874,E2 25633.874} C_VEL
LIN {X 0,Y 536.46,Z 398.914,A -85,B 0,C 180,E1 25630.396,E2 25630.396} C_VEL
LIN {X 0,Y 536.455,Z 398.886,A -85,B 0,C 180,E1 25626.956,E2 25626.956} C_VEL
LIN {X 0,Y 536.444,Z 398.909,A -85,B 0,C 180,E1 25623.545,E2 25623.545} C_VEL
LIN {X 0,Y 536.463,Z 398.911,A -85,B 0,C 180,E1 25620.074,E2 25620.074} C_VEL
LIN {X 0,Y 536.457,Z 398.909,A -85,B 0,C 180,E1 25616.615,E2 25616.615} C_VEL
LIN {X 0,Y 536.445,Z 398.91,A -85,B 0,C 180,E1 25613.25,E2 25613.25} C_VEL
LIN {X 0,Y 536.46,Z 398.909,A -85,B 0,C 180,E1 25609.833,E2 25609.833} C_VEL
LIN {X 0,Y 536.458,Z 398.9,A -85,B 0,C 180,E1 25606.316,E2 25606.316} C_VEL
LIN {X 0,Y 536.446,Z 398.905,A -85,B 0,C 180,E1 25602.903,E2 25602.903} C_VEL
LIN {X 0,Y 536.465,Z 398.912,A -85,B 0,C 180,E1 25599.461,E2 25599.461} C_VEL
LIN {X 0,Y 536.454,Z 398.901,A -85,B 0,C 180,E1 25595.952,E2 25595.952} C_VEL
LIN {X 0,Y 536.446,Z 398.905,A -85,B 0,C 180,E1 25592.592,E2 25592.592} C_VEL
LIN {X 0,Y 536.456,Z 398.91,A -85,B 0,C 180,E1 25589.231,E2 25589.231} C_VEL
LIN {X 0,Y 536.459,Z 398.897,A -85,B 0,C 180,E1 25585.739,E2 25585.739} C_VEL
LIN {X 0,Y 536.449,Z 398.909,A -85,B 0,C 180,E1 25582.348,E2 25582.348} C_VEL
LIN {X 0,Y 536.449,Z 398.904,A -85,B 0,C 180,E1 25579.037,E2 25579.037} C_VEL
LIN {X 0,Y 536.462,Z 398.902,A -85,B 0,C 180,E1 25575.569,E2 25575.569} C_VEL
LIN {X 0,Y 536.455,Z 398.913,A -85,B 0,C 180,E1 25572.159,E2 25572.159} C_VEL
LIN {X 0,Y 536.448,Z 398.903,A -85,B 0,C 180,E1 25568.792,E2 25568.792} C_VEL
LIN {X 0,Y 536.453,Z 398.906,A -85,B 0,C 180,E1 25565.455,E2 25565.455} C_VEL
LIN {X 0,Y 536.46,Z 398.907,A -85,B 0,C 180,E1 25562.03,E2 25562.03} C_VEL
LIN {X 0,Y 536.449,Z 398.904,A -85,B 0,C 180,E1 25558.612,E2 25558.612} C_VEL
LIN {X 0,Y 536.452,Z 398.908,A -85,B 0,C 180,E1 25555.189,E2 25555.189} C_VEL
LIN {X 0,Y 536.46,Z 398.906,A -85,B 0,C 180,E1 25551.749,E2 25551.749} C_VEL
LIN {X 0,Y 536.448,Z 398.904,A -85,B 0,C 180,E1 25548.279,E2 25548.279} C_VEL
LIN {X 0,Y 536.453,Z 398.908,A -85,B 0,C 180,E1 25544.875,E2 25544.875} C_VEL
LIN {X 0,Y 536.458,Z 398.912,A -85,B 0,C 180,E1 25541.415,E2 25541.415} C_VEL
LIN {X 0,Y 536.45,Z 398.906,A -85,B 0,C 180,E1 25537.999,E2 25537.999} C_VEL
LIN {X 0,Y 536.454,Z 398.91,A -85,B 0,C 180,E1 25534.616,E2 25534.616} C_VEL
LIN {X 0,Y 536.447,Z 398.909,A -85,B 0,C 180,E1 25531.258,E2 25531.258} C_VEL
LIN {X 0,Y 536.456,Z 398.903,A -85,B 0,C 180,E1 25527.788,E2 25527.788} C_VEL
LIN {X 0,Y 536.457,Z 398.912,A -85,B 0,C 180,E1 25524.354,E2 25524.354} C_VEL
LIN {X 0,Y 536.445,Z 398.912,A -85,B 0,C 180,E1 25520.951,E2 25520.951} C_VEL
LIN {X 0,Y 536.46,Z 398.907,A -85,B 0,C 180,E1 25517.568,E2 25517.568} C_VEL
LIN {X 0,Y 536.46,Z 398.911,A -85,B 0,C 180,E1 25514.147,E2 25514.147} C_VEL
LIN {X 0,Y 536.489,Z 399.11,A -85,B 0,C 180,E1 25511.282,E2 25511.282} C_VEL
LIN {X 0,Y 537.761,Z 402.414,A -85,B 0,C 180,E1 25510.881,E2 25510.881} C_VEL
LIN {X 0,Y 547.1,Z 422.785,A -85,B 0,C 180,E1 25508.706,E2 25508.706} C_VEL
LIN {X 0,Y 546.079,Z 455.645,A -85,B 0,C 180,E1 25506.579,E2 25506.579} C_VEL
LIN {X 0,Y 548.134,Z 469.076,A -85,B 0,C 180,E1 25506.204,E2 25506.204} C_VEL
LIN {X 0,Y 546.065,Z 689.19,A -85,B 0,C 180,E1 25502.916,E2 25502.916} C_VEL
LIN {X 0,Y 545.336,Z 762.473,A -85,B 0,C 180,E1 25501.809,E2 25501.809} C_VEL
LIN {X 0,Y 544.739,Z 784.112,A -85,B 0,C 180,E1 25501.285,E2 25501.285} C_VEL
LIN {X 0,Y 544.046,Z 806.179,A -85,B 0,C 180,E1 25500.543,E2 25500.543} C_VEL
LIN {X 0,Y 543.259,Z 826.357,A -85,B 0,C 180,E1 25499.677,E2 25499.677} C_VEL
LIN {X 0,Y 542.367,Z 845.73,A -85,B 0,C 180,E1 25498.642,E2 25498.642} C_VEL
LIN {X 0,Y 541.361,Z 866.179,A -85,B 0,C 180,E1 25497.331,E2 25497.331} C_VEL
LIN {X 0,Y 540.407,Z 885.087,A -85,B 0,C 180,E1 25495.892,E2 25495.892} C_VEL
LIN {X 0,Y 539.482,Z 902.887,A -85,B 0,C 180,E1 25494.297,E2 25494.297} C_VEL
LIN {X 0,Y 538.63,Z 919.163,A -85,B 0,C 180,E1 25492.599,E2 25492.599} C_VEL
LIN {X 0,Y 537.869,Z 935.009,A -85,B 0,C 180,E1 25490.685,E2 25490.685} C_VEL
LIN {X 0,Y 537.262,Z 949.195,A -85,B 0,C 180,E1 25488.692,E2 25488.692} C_VEL
LIN {X 0,Y 536.792,Z 961.451,A -85,B 0,C 180,E1 25486.671,E2 25486.671} C_VEL
LIN {X 0,Y 536.421,Z 972.807,A -85,B 0,C 180,E1 25484.466,E2 25484.466} C_VEL
LIN {X 0,Y 536.18,Z 982.252,A -85,B 0,C 180,E1 25482.275,E2 25482.275} C_VEL
LIN {X 0,Y 536.035,Z 989.877,A -85,B 0,C 180,E1 25480.1,E2 25480.1} C_VEL
LIN {X 0,Y 535.956,Z 996.14,A -85,B 0,C 180,E1 25477.829,E2 25477.829} C_VEL
LIN {X 0,Y 535.922,Z 1000.82,A -85,B 0,C 180,E1 25475.569,E2 25475.569} C_VEL
LIN {X 0,Y 535.911,Z 1003.783,A -85,B 0,C 180,E1 25473.318,E2 25473.318} C_VEL
LIN {X 0,Y 535.905,Z 1005.305,A -85,B 0,C 180,E1 25470.964,E2 25470.964} C_VEL
LIN {X 0,Y 535.907,Z 1005.238,A -85,B 0,C 180,E1 25468.719,E2 25468.719} C_VEL
LIN {X 0,Y 535.912,Z 1003.562,A -85,B 0,C 180,E1 25466.473,E2 25466.473} C_VEL
LIN {X 0,Y 535.928,Z 1000.431,A -85,B 0,C 180,E1 25464.22,E2 25464.22} C_VEL
LIN {X 0,Y 535.962,Z 995.896,A -85,B 0,C 180,E1 25462.068,E2 25462.068} C_VEL
LIN {X 0,Y 536.054,Z 989.185,A -85,B 0,C 180,E1 25459.688,E2 25459.688} C_VEL
LIN {X 0,Y 536.207,Z 981.44,A -85,B 0,C 180,E1 25457.511,E2 25457.511} C_VEL
LIN {X 0,Y 536.457,Z 971.752,A -85,B 0,C 180,E1 25455.311,E2 25455.311} C_VEL
LIN {X 0,Y 536.835,Z 960.209,A -85,B 0,C 180,E1 25453.112,E2 25453.112} C_VEL
LIN {X 0,Y 537.318,Z 947.892,A -85,B 0,C 180,E1 25451.111,E2 25451.111} C_VEL
LIN {X 0,Y 537.956,Z 933.345,A -85,B 0,C 180,E1 25449.096,E2 25449.096} C_VEL
LIN {X 0,Y 538.675,Z 918.194,A -85,B 0,C 180,E1 25447.293,E2 25447.293} C_VEL
LIN {X 0,Y 539.592,Z 900.524,A -85,B 0,C 180,E1 25445.48,E2 25445.48} C_VEL
LIN {X 0,Y 540.51,Z 883.308,A -85,B 0,C 180,E1 25443.961,E2 25443.961} C_VEL
LIN {X 0,Y 541.433,Z 864.751,A -85,B 0,C 180,E1 25442.568,E2 25442.568} C_VEL
LIN {X 0,Y 542.402,Z 844.909,A -85,B 0,C 180,E1 25441.31,E2 25441.31} C_VEL
LIN {X 0,Y 543.297,Z 825.222,A -85,B 0,C 180,E1 25440.27,E2 25440.27} C_VEL
LIN {X 0,Y 544.071,Z 805.574,A -85,B 0,C 180,E1 25439.434,E2 25439.434} C_VEL
LIN {X 0,Y 544.766,Z 783.001,A -85,B 0,C 180,E1 25438.684,E2 25438.684} C_VEL
LIN {X 0,Y 545.351,Z 761.405,A -85,B 0,C 180,E1 25438.172,E2 25438.172} C_VEL
LIN {X 0,Y 547.071,Z 579.989,A -85,B 0,C 180,E1 25435.465,E2 25435.465} C_VEL
LIN {X 0,Y 547.958,Z 466.754,A -85,B 0,C 180,E1 25433.746,E2 25433.746} C_VEL
LIN {X 0,Y 545.992,Z 454.694,A -85,B 0,C 180,E1 25433.382,E2 25433.382} C_VEL
LIN {X 0,Y 547.1,Z 422.786,A -85,B 0,C 180,E1 25431.294,E2 25431.294} C_VEL
LIN {X 0,Y 536.527,Z 399.383,A -85,B 0,C 180,E1 25428.799,E2 25428.799} C_VEL
LIN {X 0,Y 536.462,Z 398.899,A -85,B 0,C 180,E1 25428.364,E2 25428.364} C_VEL
LIN {X 0,Y 536.429,Z 398.914,A -85,B 0,C 180,E1 25425.06,E2 25425.06} C_VEL
LIN {X 0,Y 536.447,Z 398.914,A -85,B 0,C 180,E1 25421.639,E2 25421.639} C_VEL
LIN {X 0,Y 536.464,Z 398.91,A -85,B 0,C 180,E1 25418.227,E2 25418.227} C_VEL
LIN {X 0,Y 536.413,Z 398.914,A -85,B 0,C 180,E1 25414.906,E2 25414.906} C_VEL
LIN {X 0,Y 536.45,Z 398.913,A -85,B 0,C 180,E1 25411.583,E2 25411.583} C_VEL
LIN {X 0,Y 536.418,Z 398.913,A -85,B 0,C 180,E1 25408.379,E2 25408.379} C_VEL
LIN {X 0,Y 536.404,Z 398.915,A -85,B 0,C 180,E1 25405.032,E2 25405.032} C_VEL
LIN {X 0,Y 536.458,Z 398.914,A -85,B 0,C 180,E1 25401.771,E2 25401.771} C_VEL
LIN {X 0,Y 536.385,Z 398.915,A -85,B 0,C 180,E1 25398.475,E2 25398.475} C_VEL
LIN {X 0,Y 536.411,Z 398.913,A -85,B 0,C 180,E1 25395.127,E2 25395.127} C_VEL
LIN {X 0,Y 536.392,Z 398.917,A -85,B 0,C 180,E1 25392.05,E2 25392.05} C_VEL
LIN {X 0,Y 536.392,Z 398.912,A -85,B 0,C 180,E1 25388.576,E2 25388.576} C_VEL
LIN {X 0,Y 536.448,Z 398.912,A -85,B 0,C 180,E1 25385.454,E2 25385.454} C_VEL
LIN {X 0,Y 536.399,Z 398.912,A -85,B 0,C 180,E1 25382.136,E2 25382.136} C_VEL
LIN {X 0,Y 536.448,Z 398.911,A -85,B 0,C 180,E1 25378.825,E2 25378.825} C_VEL
LIN {X 0,Y 536.433,Z 398.912,A -85,B 0,C 180,E1 25375.51,E2 25375.51} C_VEL
LIN {X 0,Y 536.419,Z 398.913,A -85,B 0,C 180,E1 25372.179,E2 25372.179} C_VEL
LIN {X 0,Y 536.466,Z 398.909,A -85,B 0,C 180,E1 25368.823,E2 25368.823} C_VEL
LIN {X 0,Y 536.437,Z 398.914,A -85,B 0,C 180,E1 25365.426,E2 25365.426} C_VEL
LIN {X 0,Y 536.436,Z 398.911,A -85,B 0,C 180,E1 25361.976,E2 25361.976} C_VEL
LIN {X 0,Y 536.459,Z 398.902,A -85,B 0,C 180,E1 25358.688,E2 25358.688} C_VEL
LIN {X 0,Y 536.443,Z 398.904,A -85,B 0,C 180,E1 25355.322,E2 25355.322} C_VEL
LIN {X 0,Y 536.481,Z 399.188,A -85,B 0,C 180,E1 25353.429,E2 25353.429} C_VEL
LIN {X 0,Y 543.307,Z 416.706,A -85,B 0,C 180,E1 25351.293,E2 25351.293} C_VEL
LIN {X 0,Y 544.048,Z 419.273,A -85,B 0,C 180,E1 25351.013,E2 25351.013} C_VEL
LIN {X 0,Y 543.008,Z 443.458,A -85,B 0,C 180,E1 25349.044,E2 25349.044} C_VEL
LIN {X 0,Y 542.408,Z 449.228,A -85,B 0,C 180,E1 25348.704,E2 25348.704} C_VEL
LIN {X 0,Y 541.115,Z 456.652,A -85,B 0,C 180,E1 25348.481,E2 25348.481} C_VEL
LIN {X 0,Y 538.606,Z 471.28,A -85,B 0,C 180,E1 25348.326,E2 25348.326} C_VEL
LIN {X 0,Y 538.146,Z 478.144,A -85,B 0,C 180,E1 25348.25,E2 25348.25} C_VEL
LIN {X 0,Y 536.024,Z 700.396,A -85,B 0,C 180,E1 25344.988,E2 25344.988} C_VEL
LIN {X 0,Y 535.65,Z 721.912,A -85,B 0,C 180,E1 25344.594,E2 25344.594} C_VEL
LIN {X 0,Y 535.087,Z 742.465,A -85,B 0,C 180,E1 25344.018,E2 25344.018} C_VEL
LIN {X 0,Y 534.408,Z 762.38,A -85,B 0,C 180,E1 25343.256,E2 25343.256} C_VEL
LIN {X 0,Y 533.647,Z 780.951,A -85,B 0,C 180,E1 25342.352,E2 25342.352} C_VEL
LIN {X 0,Y 532.773,Z 800.29,A -85,B 0,C 180,E1 25341.184,E2 25341.184} C_VEL
LIN {X 0,Y 531.877,Z 818.42,A -85,B 0,C 180,E1 25339.849,E2 25339.849} C_VEL
LIN {X 0,Y 531.014,Z 835.25,A -85,B 0,C 180,E1 25338.371,E2 25338.371} C_VEL
LIN {X 0,Y 530.259,Z 850.362,A -85,B 0,C 180,E1 25336.805,E2 25336.805} C_VEL
LIN {X 0,Y 529.558,Z 865.208,A -85,B 0,C 180,E1 25334.999,E2 25334.999} C_VEL
LIN {X 0,Y 528.994,Z 878.542,A -85,B 0,C 180,E1 25333.077,E2 25333.077} C_VEL
LIN {X 0,Y 528.572,Z 890.1,A -85,B 0,C 180,E1 25331.096,E2 25331.096} C_VEL
LIN {X 0,Y 528.275,Z 899.986,A -85,B 0,C 180,E1 25329.065,E2 25329.065} C_VEL
LIN {X 0,Y 528.077,Z 908.573,A -85,B 0,C 180,E1 25326.88,E2 25326.88} C_VEL
LIN {X 0,Y 527.976,Z 915.192,A -85,B 0,C 180,E1 25324.725,E2 25324.725} C_VEL
LIN {X 0,Y 527.923,Z 920.19,A -85,B 0,C 180,E1 25322.536,E2 25322.536} C_VEL
LIN {X 0,Y 527.903,Z 923.498,A -85,B 0,C 180,E1 25320.374,E2 25320.374} C_VEL
LIN {X 0,Y 527.902,Z 925.206,A -85,B 0,C 180,E1 25318.259,E2 25318.259} C_VEL
LIN {X 0,Y 527.91,Z 925.321,A -85,B 0,C 180,E1 25316.063,E2 25316.063} C_VEL
LIN {X 0,Y 527.905,Z 923.797,A -85,B 0,C 180,E1 25313.821,E2 25313.821} C_VEL
LIN {X 0,Y 527.916,Z 920.529,A -85,B 0,C 180,E1 25311.554,E2 25311.554} C_VEL
LIN {X 0,Y 527.963,Z 915.836,A -85,B 0,C 180,E1 25309.418,E2 25309.418} C_VEL
LIN {X 0,Y 528.063,Z 909.471,A -85,B 0,C 180,E1 25307.291,E2 25307.291} C_VEL
LIN {X 0,Y 528.228,Z 901.683,A -85,B 0,C 180,E1 25305.252,E2 25305.252} C_VEL
LIN {X 0,Y 528.513,Z 891.68,A -85,B 0,C 180,E1 25303.119,E2 25303.119} C_VEL
LIN {X 0,Y 528.929,Z 880.307,A -85,B 0,C 180,E1 25301.114,E2 25301.114} C_VEL
LIN {X 0,Y 529.463,Z 867.637,A -85,B 0,C 180,E1 25299.234,E2 25299.234} C_VEL
LIN {X 0,Y 530.116,Z 853.688,A -85,B 0,C 180,E1 25297.475,E2 25297.475} C_VEL
LIN {X 0,Y 530.903,Z 837.779,A -85,B 0,C 180,E1 25295.78,E2 25295.78} C_VEL
LIN {X 0,Y 531.749,Z 820.815,A -85,B 0,C 180,E1 25294.257,E2 25294.257} C_VEL
LIN {X 0,Y 532.59,Z 803.522,A -85,B 0,C 180,E1 25292.952,E2 25292.952} C_VEL
LIN {X 0,Y 533.471,Z 784.685,A -85,B 0,C 180,E1 25291.77,E2 25291.77} C_VEL
LIN {X 0,Y 534.278,Z 765.705,A -85,B 0,C 180,E1 25290.802,E2 25290.802} C_VEL
LIN {X 0,Y 534.973,Z 746.096,A -85,B 0,C 180,E1 25290.011,E2 25290.011} C_VEL
LIN {X 0,Y 535.605,Z 725.438,A -85,B 0,C 180,E1 25289.396,E2 25289.396} C_VEL
LIN {X 0,Y 535.977,Z 704.191,A -85,B 0,C 180,E1 25288.979,E2 25288.979} C_VEL
LIN {X 0,Y 538.212,Z 467.274,A -85,B 0,C 180,E1 25285.506,E2 25285.506} C_VEL
LIN {X 0,Y 535.714,Z 452.343,A -85,B 0,C 180,E1 25285.073,E2 25285.073} C_VEL
LIN {X 0,Y 536.965,Z 422.008,A -85,B 0,C 180,E1 25282.616,E2 25282.616} C_VEL
LIN {X 0,Y 530.652,Z 405.712,A -85,B 0,C 180,E1 25280.673,E2 25280.673} C_VEL
LIN {X 0,Y 528.539,Z 400.113,A -85,B 0,C 180,E1 25279.948,E2 25279.948} C_VEL
LIN {X 0,Y 528.511,Z 399.882,A -85,B 0,C 180,E1 25276.51,E2 25276.51} C_VEL
LIN {X 0,Y 528.517,Z 399.881,A -85,B 0,C 180,E1 25273.173,E2 25273.173} C_VEL
LIN {X 0,Y 528.504,Z 399.9,A -85,B 0,C 180,E1 25269.742,E2 25269.742} C_VEL
LIN {X 0,Y 528.517,Z 399.882,A -85,B 0,C 180,E1 25266.235,E2 25266.235} C_VEL
LIN {X 0,Y 528.517,Z 399.898,A -85,B 0,C 180,E1 25262.752,E2 25262.752} C_VEL
LIN {X 0,Y 528.505,Z 399.893,A -85,B 0,C 180,E1 25259.407,E2 25259.407} C_VEL
LIN {X 0,Y 528.519,Z 399.897,A -85,B 0,C 180,E1 25255.944,E2 25255.944} C_VEL
LIN {X 0,Y 528.517,Z 399.898,A -85,B 0,C 180,E1 25252.469,E2 25252.469} C_VEL
LIN {X 0,Y 528.506,Z 399.899,A -85,B 0,C 180,E1 25249.11,E2 25249.11} C_VEL
LIN {X 0,Y 528.522,Z 399.895,A -85,B 0,C 180,E1 25245.652,E2 25245.652} C_VEL
LIN {X 0,Y 528.515,Z 399.892,A -85,B 0,C 180,E1 25242.131,E2 25242.131} C_VEL
LIN {X 0,Y 528.507,Z 399.897,A -85,B 0,C 180,E1 25238.771,E2 25238.771} C_VEL
LIN {X 0,Y 528.518,Z 399.896,A -85,B 0,C 180,E1 25235.373,E2 25235.373} C_VEL
LIN {X 0,Y 528.518,Z 399.891,A -85,B 0,C 180,E1 25231.849,E2 25231.849} C_VEL
LIN {X 0,Y 528.508,Z 399.899,A -85,B 0,C 180,E1 25228.473,E2 25228.473} C_VEL
LIN {X 0,Y 528.518,Z 399.892,A -85,B 0,C 180,E1 25225.016,E2 25225.016} C_VEL
LIN {X 0,Y 528.518,Z 399.893,A -85,B 0,C 180,E1 25221.532,E2 25221.532} C_VEL
LIN {X 0,Y 528.511,Z 399.898,A -85,B 0,C 180,E1 25218.075,E2 25218.075} C_VEL
LIN {X 0,Y 528.518,Z 399.894,A -85,B 0,C 180,E1 25214.685,E2 25214.685} C_VEL
LIN {X 0,Y 528.515,Z 399.896,A -85,B 0,C 180,E1 25211.126,E2 25211.126} C_VEL
LIN {X 0,Y 528.511,Z 399.896,A -85,B 0,C 180,E1 25207.72,E2 25207.72} C_VEL
LIN {X 0,Y 528.515,Z 399.899,A -85,B 0,C 180,E1 25204.34,E2 25204.34} C_VEL
LIN {X 0,Y 528.518,Z 399.895,A -85,B 0,C 180,E1 25200.867,E2 25200.867} C_VEL
LIN {X 0,Y 528.512,Z 399.895,A -85,B 0,C 180,E1 25197.398,E2 25197.398} C_VEL
LIN {X 0,Y 528.517,Z 399.9,A -85,B 0,C 180,E1 25193.919,E2 25193.919} C_VEL
LIN {X 0,Y 528.514,Z 399.897,A -85,B 0,C 180,E1 25190.417,E2 25190.417} C_VEL
LIN {X 0,Y 528.515,Z 399.897,A -85,B 0,C 180,E1 25186.982,E2 25186.982} C_VEL
LIN {X 0,Y 528.515,Z 399.897,A -85,B 0,C 180,E1 25183.57,E2 25183.57} C_VEL
LIN {X 0,Y 528.514,Z 399.895,A -85,B 0,C 180,E1 25180.091,E2 25180.091} C_VEL
LIN {X 0,Y 528.516,Z 399.899,A -85,B 0,C 180,E1 25176.71,E2 25176.71} C_VEL
LIN {X 0,Y 528.512,Z 399.902,A -85,B 0,C 180,E1 25173.247,E2 25173.247} C_VEL
LIN {X 0,Y 528.515,Z 399.898,A -85,B 0,C 180,E1 25169.787,E2 25169.787} C_VEL
LIN {X 0,Y 528.517,Z 399.9,A -85,B 0,C 180,E1 25166.338,E2 25166.338} C_VEL
LIN {X 0,Y 528.506,Z 399.904,A -85,B 0,C 180,E1 25162.976,E2 25162.976} C_VEL
LIN {X 0,Y 528.52,Z 399.892,A -85,B 0,C 180,E1 25159.51,E2 25159.51} C_VEL
LIN {X 0,Y 528.514,Z 399.875,A -85,B 0,C 180,E1 25156.029,E2 25156.029} C_VEL
LIN {X 0,Y 528.501,Z 399.878,A -85,B 0,C 180,E1 25152.614,E2 25152.614} C_VEL
LIN {X 0,Y 528.556,Z 400.169,A -85,B 0,C 180,E1 25151.896,E2 25151.896} C_VEL
LIN {X 0,Y 531.186,Z 406.507,A -85,B 0,C 180,E1 25151.156,E2 25151.156} C_VEL
LIN {X 0,Y 540.314,Z 426.373,A -85,B 0,C 180,E1 25149.006,E2 25149.006} C_VEL
LIN {X 0,Y 539.4,Z 455.713,A -85,B 0,C 180,E1 25147.105,E2 25147.105} C_VEL
LIN {X 0,Y 541.663,Z 470.56,A -85,B 0,C 180,E1 25146.683,E2 25146.683} C_VEL
LIN {X 0,Y 539.336,Z 690.716,A -85,B 0,C 180,E1 25143.356,E2 25143.356} C_VEL
LIN {X 0,Y 538.534,Z 762.472,A -85,B 0,C 180,E1 25142.259,E2 25142.259} C_VEL
LIN {X 0,Y 537.872,Z 784.11,A -85,B 0,C 180,E1 25141.73,E2 25141.73} C_VEL
LIN {X 0,Y 537.101,Z 806.176,A -85,B 0,C 180,E1 25140.981,E2 25140.981} C_VEL
LIN {X 0,Y 536.202,Z 826.64,A -85,B 0,C 180,E1 25140.092,E2 25140.092} C_VEL
LIN {X 0,Y 535.179,Z 846.628,A -85,B 0,C 180,E1 25139.008,E2 25139.008} C_VEL
LIN {X 0,Y 534.04,Z 867.109,A -85,B 0,C 180,E1 25137.668,E2 25137.668} C_VEL
LIN {X 0,Y 532.98,Z 885.752,A -85,B 0,C 180,E1 25136.22,E2 25136.22} C_VEL
LIN {X 0,Y 531.963,Z 903.197,A -85,B 0,C 180,E1 25134.633,E2 25134.633} C_VEL
LIN {X 0,Y 530.988,Z 919.669,A -85,B 0,C 180,E1 25132.884,E2 25132.884} C_VEL
LIN {X 0,Y 530.109,Z 935.86,A -85,B 0,C 180,E1 25130.886,E2 25130.886} C_VEL
LIN {X 0,Y 529.418,Z 950.036,A -85,B 0,C 180,E1 25128.843,E2 25128.843} C_VEL
LIN {X 0,Y 528.877,Z 962.719,A -85,B 0,C 180,E1 25126.702,E2 25126.702} C_VEL
LIN {X 0,Y 528.485,Z 973.323,A -85,B 0,C 180,E1 25124.576,E2 25124.576} C_VEL
LIN {X 0,Y 528.197,Z 983.063,A -85,B 0,C 180,E1 25122.242,E2 25122.242} C_VEL
LIN {X 0,Y 528.039,Z 990.583,A -85,B 0,C 180,E1 25120.034,E2 25120.034} C_VEL
LIN {X 0,Y 527.951,Z 996.649,A -85,B 0,C 180,E1 25117.73,E2 25117.73} C_VEL
LIN {X 0,Y 527.908,Z 1001.3,A -85,B 0,C 180,E1 25115.327,E2 25115.327} C_VEL
LIN {X 0,Y 527.903,Z 1004.008,A -85,B 0,C 180,E1 25113.151,E2 25113.151} C_VEL
LIN {X 0,Y 527.896,Z 1005.35,A -85,B 0,C 180,E1 25110.762,E2 25110.762} C_VEL
LIN {X 0,Y 527.899,Z 1005.151,A -85,B 0,C 180,E1 25108.483,E2 25108.483} C_VEL
LIN {X 0,Y 527.909,Z 1003.336,A -85,B 0,C 180,E1 25106.202,E2 25106.202} C_VEL
LIN {X 0,Y 527.933,Z 999.814,A -85,B 0,C 180,E1 25103.805,E2 25103.805} C_VEL
LIN {X 0,Y 527.987,Z 994.878,A -85,B 0,C 180,E1 25101.508,E2 25101.508} C_VEL
LIN {X 0,Y 528.091,Z 988.121,A -85,B 0,C 180,E1 25099.199,E2 25099.199} C_VEL
LIN {X 0,Y 528.293,Z 979.609,A -85,B 0,C 180,E1 25096.876,E2 25096.876} C_VEL
LIN {X 0,Y 528.617,Z 969.7,A -85,B 0,C 180,E1 25094.648,E2 25094.648} C_VEL
LIN {X 0,Y 529.053,Z 958.29,A -85,B 0,C 180,E1 25092.516,E2 25092.516} C_VEL
LIN {X 0,Y 529.665,Z 944.809,A -85,B 0,C 180,E1 25090.369,E2 25090.369} C_VEL
LIN {X 0,Y 530.4,Z 930.678,A -85,B 0,C 180,E1 25088.436,E2 25088.436} C_VEL
LIN {X 0,Y 531.291,Z 914.839,A -85,B 0,C 180,E1 25086.571,E2 25086.571} C_VEL
LIN {X 0,Y 532.24,Z 898.092,A -85,B 0,C 180,E1 25084.881,E2 25084.881} C_VEL
LIN {X 0,Y 533.335,Z 879.439,A -85,B 0,C 180,E1 25083.264,E2 25083.264} C_VEL
LIN {X 0,Y 534.442,Z 860.595,A -85,B 0,C 180,E1 25081.875,E2 25081.875} C_VEL
LIN {X 0,Y 535.46,Z 840.894,A -85,B 0,C 180,E1 25080.658,E2 25080.658} C_VEL
LIN {X 0,Y 536.46,Z 821.02,A -85,B 0,C 180,E1 25079.648,E2 25079.648} C_VEL
LIN {X 0,Y 537.337,Z 800.476,A -85,B 0,C 180,E1 25078.798,E2 25078.798} C_VEL
LIN {X 0,Y 538.045,Z 779.484,A -85,B 0,C 180,E1 25078.142,E2 25078.142} C_VEL
LIN {X 0,Y 538.602,Z 757.084,A -85,B 0,C 180,E1 25077.646,E2 25077.646} C_VEL
LIN {X 0,Y 540.94,Z 536.857,A -85,B 0,C 180,E1 25074.329,E2 25074.329} C_VEL
LIN {X 0,Y 541.497,Z 468.241,A -85,B 0,C 180,E1 25073.267,E2 25073.267} C_VEL
LIN {X 0,Y 539.306,Z 454.896,A -85,B 0,C 180,E1 25072.864,E2 25072.864} C_VEL
LIN {X 0,Y 540.13,Z 425.748,A -85,B 0,C 180,E1 25070.946,E2 25070.946} C_VEL
LIN {X 0,Y 528.594,Z 400.356,A -85,B 0,C 180,E1 25068.182,E2 25068.182} C_VEL
LIN {X 0,Y 528.507,Z 399.899,A -85,B 0,C 180,E1 25067.667,E2 25067.667} C_VEL
LIN {X 0,Y 528.526,Z 399.902,A -85,B 0,C 180,E1 25064.199,E2 25064.199} C_VEL
LIN {X 0,Y 528.49,Z 399.902,A -85,B 0,C 180,E1 25060.826,E2 25060.826} C_VEL
LIN {X 0,Y 528.49,Z 399.905,A -85,B 0,C 180,E1 25057.388,E2 25057.388} C_VEL
LIN {X 0,Y 528.525,Z 399.899,A -85,B 0,C 180,E1 25054.051,E2 25054.051} C_VEL
LIN {X 0,Y 528.469,Z 399.904,A -85,B 0,C 180,E1 25050.719,E2 25050.719} C_VEL
LIN {X 0,Y 528.49,Z 399.901,A -85,B 0,C 180,E1 25047.37,E2 25047.37} C_VEL
LIN {X 0,Y 528.484,Z 399.903,A -85,B 0,C 180,E1 25044.12,E2 25044.12} C_VEL
LIN {X 0,Y 528.454,Z 399.902,A -85,B 0,C 180,E1 25040.836,E2 25040.836} C_VEL
LIN {X 0,Y 528.513,Z 399.9,A -85,B 0,C 180,E1 25037.558,E2 25037.558} C_VEL
LIN {X 0,Y 528.44,Z 399.902,A -85,B 0,C 180,E1 25034.351,E2 25034.351} C_VEL
LIN {X 0,Y 528.476,Z 399.905,A -85,B 0,C 180,E1 25031.016,E2 25031.016} C_VEL
LIN {X 0,Y 528.471,Z 399.901,A -85,B 0,C 180,E1 25027.829,E2 25027.829} C_VEL
LIN {X 0,Y 528.459,Z 399.903,A -85,B 0,C 180,E1 25024.42,E2 25024.42} C_VEL
LIN {X 0,Y 528.525,Z 399.902,A -85,B 0,C 180,E1 25021.084,E2 25021.084} C_VEL
LIN {X 0,Y 528.473,Z 399.904,A -85,B 0,C 180,E1 25017.831,E2 25017.831} C_VEL
LIN {X 0,Y 528.481,Z 399.901,A -85,B 0,C 180,E1 25014.321,E2 25014.321} C_VEL
LIN {X 0,Y 528.525,Z 399.899,A -85,B 0,C 180,E1 25011.076,E2 25011.076} C_VEL
LIN {X 0,Y 528.484,Z 399.902,A -85,B 0,C 180,E1 25007.766,E2 25007.766} C_VEL
LIN {X 0,Y 528.514,Z 399.898,A -85,B 0,C 180,E1 25004.338,E2 25004.338} C_VEL
LIN {X 0,Y 528.525,Z 399.9,A -85,B 0,C 180,E1 25000.896,E2 25000.896} C_VEL
LIN {X 0,Y 528.498,Z 399.892,A -85,B 0,C 180,E1 24997.532,E2 24997.532} C_VEL
LIN {X 0,Y 528.552,Z 400.122,A -85,B 0,C 180,E1 24994.063,E2 24994.063} C_VEL
LIN {X 0,Y 530.926,Z 406.275,A -85,B 0,C 180,E1 24993.25,E2 24993.25} C_VEL
LIN {X 0,Y 537.042,Z 421.871,A -85,B 0,C 180,E1 24991.353,E2 24991.353} C_VEL
LIN {X 0,Y 535.847,Z 452.765,A -85,B 0,C 180,E1 24988.838,E2 24988.838} C_VEL
LIN {X 0,Y 538.275,Z 467.291,A -85,B 0,C 180,E1 24988.415,E2 24988.415} C_VEL
LIN {X 0,Y 538.146,Z 478.144,A -85,B 0,C 180,E1 24988.25,E2 24988.25} C_VEL
LIN {X 0,Y 537.223,Z 485.84,A -85,B 0,C 180,E1 24988.195,E2 24988.195} C_VEL
LIN {X 0,Y 531.786,Z 506.374,A -85,B 0,C 180,E1 24988.263,E2 24988.263} C_VEL
LIN {X 0,Y 531.103,Z 512.976,A -85,B 0,C 180,E1 24988.208,E2 24988.208} C_VEL
LIN {X 0,Y 528.777,Z 714.373,A -85,B 0,C 180,E1 24985.165,E2 24985.165} C_VEL
LIN {X 0,Y 528.169,Z 736.078,A -85,B 0,C 180,E1 24984.624,E2 24984.624} C_VEL
LIN {X 0,Y 527.47,Z 755.297,A -85,B 0,C 180,E1 24983.944,E2 24983.944} C_VEL
LIN {X 0,Y 526.626,Z 774.677,A -85,B 0,C 180,E1 24983.058,E2 24983.058} C_VEL
LIN {X 0,Y 525.651,Z 794.155,A -85,B 0,C 180,E1 24981.945,E2 24981.945} C_VEL
LIN {X 0,Y 524.701,Z 812.283,A -85,B 0,C 180,E1 24980.678,E2 24980.678} C_VEL
LIN {X 0,Y 523.748,Z 829.506,A -85,B 0,C 180,E1 24979.239,E2 24979.239} C_VEL
LIN {X 0,Y 522.851,Z 845.463,A -85,B 0,C 180,E1 24977.659,E2 24977.659} C_VEL
LIN {X 0,Y 522.032,Z 860.436,A -85,B 0,C 180,E1 24975.905,E2 24975.905} C_VEL
LIN {X 0,Y 521.375,Z 873.441,A -85,B 0,C 180,E1 24974.113,E2 24974.113} C_VEL
LIN {X 0,Y 520.854,Z 885.345,A -85,B 0,C 180,E1 24972.184,E2 24972.184} C_VEL
LIN {X 0,Y 520.457,Z 895.996,A -85,B 0,C 180,E1 24970.128,E2 24970.128} C_VEL
LIN {X 0,Y 520.182,Z 905.096,A -85,B 0,C 180,E1 24967.994,E2 24967.994} C_VEL
LIN {X 0,Y 520.026,Z 912.658,A -85,B 0,C 180,E1 24965.764,E2 24965.764} C_VEL
LIN {X 0,Y 519.949,Z 918.452,A -85,B 0,C 180,E1 24963.493,E2 24963.493} C_VEL
LIN {X 0,Y 519.917,Z 922.399,A -85,B 0,C 180,E1 24961.277,E2 24961.277} C_VEL
LIN {X 0,Y 519.916,Z 924.796,A -85,B 0,C 180,E1 24958.952,E2 24958.952} C_VEL
LIN {X 0,Y 519.909,Z 925.461,A -85,B 0,C 180,E1 24956.741,E2 24956.741} C_VEL
LIN {X 0,Y 519.91,Z 924.454,A -85,B 0,C 180,E1 24954.42,E2 24954.42} C_VEL
LIN {X 0,Y 519.927,Z 921.686,A -85,B 0,C 180,E1 24952.14,E2 24952.14} C_VEL
LIN {X 0,Y 519.955,Z 917.528,A -85,B 0,C 180,E1 24950.013,E2 24950.013} C_VEL
LIN {X 0,Y 520.038,Z 911.553,A -85,B 0,C 180,E1 24947.797,E2 24947.797} C_VEL
LIN {X 0,Y 520.213,Z 904.052,A -85,B 0,C 180,E1 24945.648,E2 24945.648} C_VEL
LIN {X 0,Y 520.502,Z 894.928,A -85,B 0,C 180,E1 24943.551,E2 24943.551} C_VEL
LIN {X 0,Y 520.91,Z 884.141,A -85,B 0,C 180,E1 24941.512,E2 24941.512} C_VEL
LIN {X 0,Y 521.441,Z 872.106,A -85,B 0,C 180,E1 24939.6,E2 24939.6} C_VEL
LIN {X 0,Y 522.156,Z 857.968,A -85,B 0,C 180,E1 24937.701,E2 24937.701} C_VEL
LIN {X 0,Y 522.976,Z 842.843,A -85,B 0,C 180,E1 24935.978,E2 24935.978} C_VEL
LIN {X 0,Y 523.887,Z 826.837,A -85,B 0,C 180,E1 24934.431,E2 24934.431} C_VEL
LIN {X 0,Y 524.884,Z 809.272,A -85,B 0,C 180,E1 24933,E2 24933} C_VEL
LIN {X 0,Y 525.861,Z 790.626,A -85,B 0,C 180,E1 24931.741,E2 24931.741} C_VEL
LIN {X 0,Y 526.762,Z 771.795,A -85,B 0,C 180,E1 24930.705,E2 24930.705} C_VEL
LIN {X 0,Y 527.572,Z 752.626,A -85,B 0,C 180,E1 24929.862,E2 24929.862} C_VEL
LIN {X 0,Y 528.267,Z 732.081,A -85,B 0,C 180,E1 24929.174,E2 24929.174} C_VEL
LIN {X 0,Y 528.806,Z 711.691,A -85,B 0,C 180,E1 24928.698,E2 24928.698} C_VEL
LIN {X 0,Y 531.53,Z 467.466,A -85,B 0,C 180,E1 24925.027,E2 24925.027} C_VEL
LIN {X 0,Y 528.751,Z 452.088,A -85,B 0,C 180,E1 24924.545,E2 24924.545} C_VEL
LIN {X 0,Y 529.849,Z 424.866,A -85,B 0,C 180,E1 24922.298,E2 24922.298} C_VEL
LIN {X 0,Y 523.192,Z 407.682,A -85,B 0,C 180,E1 24920.205,E2 24920.205} C_VEL
LIN {X 0,Y 520.611,Z 401.105,A -85,B 0,C 180,E1 24919.331,E2 24919.331} C_VEL
LIN {X 0,Y 520.565,Z 400.879,A -85,B 0,C 180,E1 24915.993,E2 24915.993} C_VEL
LIN {X 0,Y 520.581,Z 400.864,A -85,B 0,C 180,E1 24912.563,E2 24912.563} C_VEL
LIN {X 0,Y 520.58,Z 400.887,A -85,B 0,C 180,E1 24909.067,E2 24909.067} C_VEL
LIN {X 0,Y 520.566,Z 400.885,A -85,B 0,C 180,E1 24905.608,E2 24905.608} C_VEL
LIN {X 0,Y 520.582,Z 400.887,A -85,B 0,C 180,E1 24902.068,E2 24902.068} C_VEL
LIN {X 0,Y 520.579,Z 400.881,A -85,B 0,C 180,E1 24898.633,E2 24898.633} C_VEL
LIN {X 0,Y 520.567,Z 400.88,A -85,B 0,C 180,E1 24895.217,E2 24895.217} C_VEL
LIN {X 0,Y 520.585,Z 400.884,A -85,B 0,C 180,E1 24891.771,E2 24891.771} C_VEL
LIN {X 0,Y 520.579,Z 400.886,A -85,B 0,C 180,E1 24888.344,E2 24888.344} C_VEL
LIN {X 0,Y 520.57,Z 400.886,A -85,B 0,C 180,E1 24884.866,E2 24884.866} C_VEL
LIN {X 0,Y 520.583,Z 400.883,A -85,B 0,C 180,E1 24881.324,E2 24881.324} C_VEL
LIN {X 0,Y 520.575,Z 400.886,A -85,B 0,C 180,E1 24877.869,E2 24877.869} C_VEL
LIN {X 0,Y 520.575,Z 400.886,A -85,B 0,C 180,E1 24874.38,E2 24874.38} C_VEL
LIN {X 0,Y 520.577,Z 400.883,A -85,B 0,C 180,E1 24870.845,E2 24870.845} C_VEL
LIN {X 0,Y 520.573,Z 400.887,A -85,B 0,C 180,E1 24867.45,E2 24867.45} C_VEL
LIN {X 0,Y 520.576,Z 400.884,A -85,B 0,C 180,E1 24864.028,E2 24864.028} C_VEL
LIN {X 0,Y 520.577,Z 400.879,A -85,B 0,C 180,E1 24860.461,E2 24860.461} C_VEL
LIN {X 0,Y 520.573,Z 400.889,A -85,B 0,C 180,E1 24856.959,E2 24856.959} C_VEL
LIN {X 0,Y 520.583,Z 400.879,A -85,B 0,C 180,E1 24853.439,E2 24853.439} C_VEL
LIN {X 0,Y 520.573,Z 400.882,A -85,B 0,C 180,E1 24849.955,E2 24849.955} C_VEL
LIN {X 0,Y 520.573,Z 400.887,A -85,B 0,C 180,E1 24846.507,E2 24846.507} C_VEL
LIN {X 0,Y 520.578,Z 400.873,A -85,B 0,C 180,E1 24842.973,E2 24842.973} C_VEL
LIN {X 0,Y 520.574,Z 400.885,A -85,B 0,C 180,E1 24839.56,E2 24839.56} C_VEL
LIN {X 0,Y 520.571,Z 400.886,A -85,B 0,C 180,E1 24836.146,E2 24836.146} C_VEL
LIN {X 0,Y 520.579,Z 400.874,A -85,B 0,C 180,E1 24832.607,E2 24832.607} C_VEL
LIN {X 0,Y 520.576,Z 400.884,A -85,B 0,C 180,E1 24829.151,E2 24829.151} C_VEL
LIN {X 0,Y 520.577,Z 400.89,A -85,B 0,C 180,E1 24825.655,E2 24825.655} C_VEL
LIN {X 0,Y 520.572,Z 400.884,A -85,B 0,C 180,E1 24822.103,E2 24822.103} C_VEL
LIN {X 0,Y 520.577,Z 400.885,A -85,B 0,C 180,E1 24818.676,E2 24818.676} C_VEL
LIN {X 0,Y 520.576,Z 400.885,A -85,B 0,C 180,E1 24815.247,E2 24815.247} C_VEL
LIN {X 0,Y 520.569,Z 400.884,A -85,B 0,C 180,E1 24811.679,E2 24811.679} C_VEL
LIN {X 0,Y 520.579,Z 400.882,A -85,B 0,C 180,E1 24808.247,E2 24808.247} C_VEL
LIN {X 0,Y 520.581,Z 400.886,A -85,B 0,C 180,E1 24804.716,E2 24804.716} C_VEL
LIN {X 0,Y 520.565,Z 400.888,A -85,B 0,C 180,E1 24801.233,E2 24801.233} C_VEL
LIN {X 0,Y 520.58,Z 400.887,A -85,B 0,C 180,E1 24797.85,E2 24797.85} C_VEL
LIN {X 0,Y 520.581,Z 400.882,A -85,B 0,C 180,E1 24794.358,E2 24794.358} C_VEL
LIN {X 0,Y 520.598,Z 401.105,A -85,B 0,C 180,E1 24792.572,E2 24792.572} C_VEL
LIN {X 0,Y 521.911,Z 404.378,A -85,B 0,C 180,E1 24792.15,E2 24792.15} C_VEL
LIN {X 0,Y 533.508,Z 429.679,A -85,B 0,C 180,E1 24789.323,E2 24789.323} C_VEL
LIN {X 0,Y 532.68,Z 455.609,A -85,B 0,C 180,E1 24787.641,E2 24787.641} C_VEL
LIN {X 0,Y 535.232,Z 471.976,A -85,B 0,C 180,E1 24787.174,E2 24787.174} C_VEL
LIN {X 0,Y 532.642,Z 692.116,A -85,B 0,C 180,E1 24783.809,E2 24783.809} C_VEL
LIN {X 0,Y 531.766,Z 762.472,A -85,B 0,C 180,E1 24782.72,E2 24782.72} C_VEL
LIN {X 0,Y 531.046,Z 784.107,A -85,B 0,C 180,E1 24782.187,E2 24782.187} C_VEL
LIN {X 0,Y 530.188,Z 806.173,A -85,B 0,C 180,E1 24781.43,E2 24781.43} C_VEL
LIN {X 0,Y 529.216,Z 826.354,A -85,B 0,C 180,E1 24780.547,E2 24780.547} C_VEL
LIN {X 0,Y 528.047,Z 846.852,A -85,B 0,C 180,E1 24779.424,E2 24779.424} C_VEL
LIN {X 0,Y 526.795,Z 867.105,A -85,B 0,C 180,E1 24778.082,E2 24778.082} C_VEL
LIN {X 0,Y 525.616,Z 885.788,A -85,B 0,C 180,E1 24776.612,E2 24776.612} C_VEL
LIN {X 0,Y 524.46,Z 903.494,A -85,B 0,C 180,E1 24774.98,E2 24774.98} C_VEL
LIN {X 0,Y 523.399,Z 919.626,A -85,B 0,C 180,E1 24773.24,E2 24773.24} C_VEL
LIN {X 0,Y 522.409,Z 935.858,A -85,B 0,C 180,E1 24771.209,E2 24771.209} C_VEL
LIN {X 0,Y 521.625,Z 950.038,A -85,B 0,C 180,E1 24769.136,E2 24769.136} C_VEL
LIN {X 0,Y 521.013,Z 962.718,A -85,B 0,C 180,E1 24766.962,E2 24766.962} C_VEL
LIN {X 0,Y 520.568,Z 973.322,A -85,B 0,C 180,E1 24764.802,E2 24764.802} C_VEL
LIN {X 0,Y 520.245,Z 983.064,A -85,B 0,C 180,E1 24762.432,E2 24762.432} C_VEL
LIN {X 0,Y 520.063,Z 990.71,A -85,B 0,C 180,E1 24760.149,E2 24760.149} C_VEL
LIN {X 0,Y 519.965,Z 996.649,A -85,B 0,C 180,E1 24757.849,E2 24757.849} C_VEL
LIN {X 0,Y 519.913,Z 1001.3,A -85,B 0,C 180,E1 24755.409,E2 24755.409} C_VEL
LIN {X 0,Y 519.905,Z 1004.008,A -85,B 0,C 180,E1 24753.199,E2 24753.199} C_VEL
LIN {X 0,Y 519.897,Z 1005.35,A -85,B 0,C 180,E1 24750.774,E2 24750.774} C_VEL
LIN {X 0,Y 519.899,Z 1005.151,A -85,B 0,C 180,E1 24748.46,E2 24748.46} C_VEL
LIN {X 0,Y 519.91,Z 1003.335,A -85,B 0,C 180,E1 24746.143,E2 24746.143} C_VEL
LIN {X 0,Y 519.938,Z 999.814,A -85,B 0,C 180,E1 24743.71,E2 24743.71} C_VEL
LIN {X 0,Y 519.993,Z 994.878,A -85,B 0,C 180,E1 24741.377,E2 24741.377} C_VEL
LIN {X 0,Y 520.115,Z 988.122,A -85,B 0,C 180,E1 24739.032,E2 24739.032} C_VEL
LIN {X 0,Y 520.348,Z 979.608,A -85,B 0,C 180,E1 24736.671,E2 24736.671} C_VEL
LIN {X 0,Y 520.717,Z 969.699,A -85,B 0,C 180,E1 24734.409,E2 24734.409} C_VEL
LIN {X 0,Y 521.212,Z 958.292,A -85,B 0,C 180,E1 24732.244,E2 24732.244} C_VEL
LIN {X 0,Y 521.903,Z 944.807,A -85,B 0,C 180,E1 24730.065,E2 24730.065} C_VEL
LIN {X 0,Y 522.734,Z 930.46,A -85,B 0,C 180,E1 24728.076,E2 24728.076} C_VEL
LIN {X 0,Y 523.739,Z 914.645,A -85,B 0,C 180,E1 24726.189,E2 24726.189} C_VEL
LIN {X 0,Y 524.831,Z 897.654,A -85,B 0,C 180,E1 24724.457,E2 24724.457} C_VEL
LIN {X 0,Y 526.042,Z 878.85,A -85,B 0,C 180,E1 24722.814,E2 24722.814} C_VEL
LIN {X 0,Y 527.293,Z 859.678,A -85,B 0,C 180,E1 24721.395,E2 24721.395} C_VEL
LIN {X 0,Y 528.383,Z 840.791,A -85,B 0,C 180,E1 24720.22,E2 24720.22} C_VEL
LIN {X 0,Y 529.521,Z 820.11,A -85,B 0,C 180,E1 24719.163,E2 24719.163} C_VEL
LIN {X 0,Y 530.485,Z 799.293,A -85,B 0,C 180,E1 24718.305,E2 24718.305} C_VEL
LIN {X 0,Y 531.263,Z 778.686,A -85,B 0,C 180,E1 24717.662,E2 24717.662} C_VEL
LIN {X 0,Y 531.853,Z 756.419,A -85,B 0,C 180,E1 24717.172,E2 24717.172} C_VEL
LIN {X 0,Y 534.437,Z 537.493,A -85,B 0,C 180,E1 24713.837,E2 24713.837} C_VEL
LIN {X 0,Y 535.071,Z 469.708,A -85,B 0,C 180,E1 24712.776,E2 24712.776} C_VEL
LIN {X 0,Y 532.579,Z 454.868,A -85,B 0,C 180,E1 24712.334,E2 24712.334} C_VEL
LIN {X 0,Y 533.425,Z 429.66,A -85,B 0,C 180,E1 24710.692,E2 24710.692} C_VEL
LIN {X 0,Y 521.722,Z 404.122,A -85,B 0,C 180,E1 24707.873,E2 24707.873} C_VEL
LIN {X 0,Y 520.592,Z 401.133,A -85,B 0,C 180,E1 24707.485,E2 24707.485} C_VEL
LIN {X 0,Y 520.588,Z 400.891,A -85,B 0,C 180,E1 24704.355,E2 24704.355} C_VEL
LIN {X 0,Y 520.548,Z 400.892,A -85,B 0,C 180,E1 24700.918,E2 24700.918} C_VEL
LIN {X 0,Y 520.559,Z 400.894,A -85,B 0,C 180,E1 24697.508,E2 24697.508} C_VEL
LIN {X 0,Y 520.583,Z 400.887,A -85,B 0,C 180,E1 24694.113,E2 24694.113} C_VEL
LIN {X 0,Y 520.529,Z 400.893,A -85,B 0,C 180,E1 24690.846,E2 24690.846} C_VEL
LIN {X 0,Y 520.561,Z 400.89,A -85,B 0,C 180,E1 24687.463,E2 24687.463} C_VEL
LIN {X 0,Y 520.541,Z 400.892,A -85,B 0,C 180,E1 24684.173,E2 24684.173} C_VEL
LIN {X 0,Y 520.515,Z 400.891,A -85,B 0,C 180,E1 24680.816,E2 24680.816} C_VEL
LIN {X 0,Y 520.574,Z 400.888,A -85,B 0,C 180,E1 24677.55,E2 24677.55} C_VEL
LIN {X 0,Y 520.505,Z 400.891,A -85,B 0,C 180,E1 24674.234,E2 24674.234} C_VEL
LIN {X 0,Y 520.516,Z 400.894,A -85,B 0,C 180,E1 24670.738,E2 24670.738} C_VEL
LIN {X 0,Y 520.579,Z 400.889,A -85,B 0,C 180,E1 24667.393,E2 24667.393} C_VEL
LIN {X 0,Y 520.521,Z 400.893,A -85,B 0,C 180,E1 24664.075,E2 24664.075} C_VEL
LIN {X 0,Y 520.546,Z 400.892,A -85,B 0,C 180,E1 24660.66,E2 24660.66} C_VEL
LIN {X 0,Y 520.572,Z 400.894,A -85,B 0,C 180,E1 24657.358,E2 24657.358} C_VEL
LIN {X 0,Y 520.536,Z 400.892,A -85,B 0,C 180,E1 24653.935,E2 24653.935} C_VEL
LIN {X 0,Y 520.567,Z 400.889,A -85,B 0,C 180,E1 24650.492,E2 24650.492} C_VEL
LIN {X 0,Y 520.581,Z 400.891,A -85,B 0,C 180,E1 24647.126,E2 24647.126} C_VEL
LIN {X 0,Y 520.551,Z 400.891,A -85,B 0,C 180,E1 24643.714,E2 24643.714} C_VEL
LIN {X 0,Y 520.579,Z 400.889,A -85,B 0,C 180,E1 24640.23,E2 24640.23} C_VEL
LIN {X 0,Y 520.585,Z 400.89,A -85,B 0,C 180,E1 24636.813,E2 24636.813} C_VEL
LIN {X 0,Y 520.613,Z 401.112,A -85,B 0,C 180,E1 24634.708,E2 24634.708} C_VEL
LIN {X 0,Y 528.579,Z 420.887,A -85,B 0,C 180,E1 24632.145,E2 24632.145} C_VEL
LIN {X 0,Y 530.186,Z 425.911,A -85,B 0,C 180,E1 24631.563,E2 24631.563} C_VEL
LIN {X 0,Y 528.965,Z 452.868,A -85,B 0,C 180,E1 24629.359,E2 24629.359} C_VEL
LIN {X 0,Y 531.679,Z 468.762,A -85,B 0,C 180,E1 24628.884,E2 24628.884} C_VEL
LIN {X 0,Y 531.103,Z 512.976,A -85,B 0,C 180,E1 24628.208,E2 24628.208} C_VEL
LIN {X 0,Y 530.2,Z 520.67,A -85,B 0,C 180,E1 24628.15,E2 24628.15} C_VEL
LIN {X 0,Y 524.729,Z 541.2,A -85,B 0,C 180,E1 24628.221,E2 24628.221} C_VEL
LIN {X 0,Y 524.024,Z 547.804,A -85,B 0,C 180,E1 24628.166,E2 24628.166} C_VEL
LIN {X 0,Y 521.884,Z 714.677,A -85,B 0,C 180,E1 24625.608,E2 24625.608} C_VEL
LIN {X 0,Y 521.223,Z 735.44,A -85,B 0,C 180,E1 24625.084,E2 24625.084} C_VEL
LIN {X 0,Y 520.438,Z 754.559,A -85,B 0,C 180,E1 24624.4,E2 24624.4} C_VEL
LIN {X 0,Y 519.451,Z 773.907,A -85,B 0,C 180,E1 24623.503,E2 24623.503} C_VEL
LIN {X 0,Y 518.36,Z 793.263,A -85,B 0,C 180,E1 24622.381,E2 24622.381} C_VEL
LIN {X 0,Y 517.35,Z 810.902,A -85,B 0,C 180,E1 24621.15,E2 24621.15} C_VEL
LIN {X 0,Y 516.27,Z 828.322,A -85,B 0,C 180,E1 24619.695,E2 24619.695} C_VEL
LIN {X 0,Y 515.256,Z 844.401,A -85,B 0,C 180,E1 24618.093,E2 24618.093} C_VEL
LIN {X 0,Y 514.369,Z 859.133,A -85,B 0,C 180,E1 24616.364,E2 24616.364} C_VEL
LIN {X 0,Y 513.603,Z 872.73,A -85,B 0,C 180,E1 24614.489,E2 24614.489} C_VEL
LIN {X 0,Y 512.972,Z 885.457,A -85,B 0,C 180,E1 24612.403,E2 24612.403} C_VEL
LIN {X 0,Y 512.523,Z 896.204,A -85,B 0,C 180,E1 24610.289,E2 24610.289} C_VEL
LIN {X 0,Y 512.215,Z 905.25,A -85,B 0,C 180,E1 24608.124,E2 24608.124} C_VEL
LIN {X 0,Y 512.039,Z 912.8,A -85,B 0,C 180,E1 24605.856,E2 24605.856} C_VEL
LIN {X 0,Y 511.955,Z 918.257,A -85,B 0,C 180,E1 24603.683,E2 24603.683} C_VEL
LIN {X 0,Y 511.918,Z 922.318,A -85,B 0,C 180,E1 24601.402,E2 24601.402} C_VEL
LIN {X 0,Y 511.911,Z 924.726,A -85,B 0,C 180,E1 24599.097,E2 24599.097} C_VEL
LIN {X 0,Y 511.912,Z 925.476,A -85,B 0,C 180,E1 24596.816,E2 24596.816} C_VEL
LIN {X 0,Y 511.912,Z 924.587,A -85,B 0,C 180,E1 24594.581,E2 24594.581} C_VEL
LIN {X 0,Y 511.923,Z 922.14,A -85,B 0,C 180,E1 24592.384,E2 24592.384} C_VEL
LIN {X 0,Y 511.959,Z 917.854,A -85,B 0,C 180,E1 24590.049,E2 24590.049} C_VEL
LIN {X 0,Y 512.046,Z 912.165,A -85,B 0,C 180,E1 24587.85,E2 24587.85} C_VEL
LIN {X 0,Y 512.239,Z 904.664,A -85,B 0,C 180,E1 24585.624,E2 24585.624} C_VEL
LIN {X 0,Y 512.562,Z 895.293,A -85,B 0,C 180,E1 24583.42,E2 24583.42} C_VEL
LIN {X 0,Y 513.016,Z 884.589,A -85,B 0,C 180,E1 24581.35,E2 24581.35} C_VEL
LIN {X 0,Y 513.607,Z 872.645,A -85,B 0,C 180,E1 24579.409,E2 24579.409} C_VEL
LIN {X 0,Y 514.397,Z 858.611,A -85,B 0,C 180,E1 24577.48,E2 24577.48} C_VEL
LIN {X 0,Y 515.304,Z 843.602,A -85,B 0,C 180,E1 24575.732,E2 24575.732} C_VEL
LIN {X 0,Y 516.297,Z 827.821,A -85,B 0,C 180,E1 24574.17,E2 24574.17} C_VEL
LIN {X 0,Y 517.39,Z 810.282,A -85,B 0,C 180,E1 24572.711,E2 24572.711} C_VEL
LIN {X 0,Y 518.456,Z 791.79,A -85,B 0,C 180,E1 24571.434,E2 24571.434} C_VEL
LIN {X 0,Y 519.531,Z 772.342,A -85,B 0,C 180,E1 24570.328,E2 24570.328} C_VEL
LIN {X 0,Y 520.488,Z 752.855,A -85,B 0,C 180,E1 24569.447,E2 24569.447} C_VEL
LIN {X 0,Y 521.284,Z 732.42,A -85,B 0,C 180,E1 24568.748,E2 24568.748} C_VEL
LIN {X 0,Y 521.878,Z 712.002,A -85,B 0,C 180,E1 24568.262,E2 24568.262} C_VEL
LIN {X 0,Y 524.916,Z 468.992,A -85,B 0,C 180,E1 24564.56,E2 24564.56} C_VEL
LIN {X 0,Y 521.844,Z 451.876,A -85,B 0,C 180,E1 24564.004,E2 24564.004} C_VEL
LIN {X 0,Y 522.964,Z 428.339,A -85,B 0,C 180,E1 24562.044,E2 24562.044} C_VEL
LIN {X 0,Y 516.448,Z 411.592,A -85,B 0,C 180,E1 24559.963,E2 24559.963} C_VEL
LIN {X 0,Y 512.668,Z 402.085,A -85,B 0,C 180,E1 24558.691,E2 24558.691} C_VEL
LIN {X 0,Y 512.645,Z 401.877,A -85,B 0,C 180,E1 24555.31,E2 24555.31} C_VEL
LIN {X 0,Y 512.626,Z 401.86,A -85,B 0,C 180,E1 24551.814,E2 24551.814} C_VEL
LIN {X 0,Y 512.644,Z 401.855,A -85,B 0,C 180,E1 24548.367,E2 24548.367} C_VEL
LIN {X 0,Y 512.64,Z 401.874,A -85,B 0,C 180,E1 24544.823,E2 24544.823} C_VEL
LIN {X 0,Y 512.634,Z 401.876,A -85,B 0,C 180,E1 24541.325,E2 24541.325} C_VEL
LIN {X 0,Y 512.637,Z 401.88,A -85,B 0,C 180,E1 24537.826,E2 24537.826} C_VEL
LIN {X 0,Y 512.638,Z 401.87,A -85,B 0,C 180,E1 24534.324,E2 24534.324} C_VEL
LIN {X 0,Y 512.643,Z 401.865,A -85,B 0,C 180,E1 24530.806,E2 24530.806} C_VEL
LIN {X 0,Y 512.631,Z 401.87,A -85,B 0,C 180,E1 24527.335,E2 24527.335} C_VEL
LIN {X 0,Y 512.64,Z 401.879,A -85,B 0,C 180,E1 24523.807,E2 24523.807} C_VEL
LIN {X 0,Y 512.646,Z 401.871,A -85,B 0,C 180,E1 24520.21,E2 24520.21} C_VEL
LIN {X 0,Y 512.629,Z 401.868,A -85,B 0,C 180,E1 24516.712,E2 24516.712} C_VEL
LIN {X 0,Y 512.645,Z 401.879,A -85,B 0,C 180,E1 24513.203,E2 24513.203} C_VEL
LIN {X 0,Y 512.638,Z 401.871,A -85,B 0,C 180,E1 24509.697,E2 24509.697} C_VEL
LIN {X 0,Y 512.632,Z 401.864,A -85,B 0,C 180,E1 24506.28,E2 24506.28} C_VEL
LIN {X 0,Y 512.645,Z 401.879,A -85,B 0,C 180,E1 24502.699,E2 24502.699} C_VEL
LIN {X 0,Y 512.633,Z 401.866,A -85,B 0,C 180,E1 24499.246,E2 24499.246} C_VEL
LIN {X 0,Y 512.64,Z 401.869,A -85,B 0,C 180,E1 24495.731,E2 24495.731} C_VEL
LIN {X 0,Y 512.639,Z 401.88,A -85,B 0,C 180,E1 24492.16,E2 24492.16} C_VEL
LIN {X 0,Y 512.633,Z 401.868,A -85,B 0,C 180,E1 24488.638,E2 24488.638} C_VEL
LIN {X 0,Y 512.643,Z 401.872,A -85,B 0,C 180,E1 24485.148,E2 24485.148} C_VEL
LIN {X 0,Y 512.636,Z 401.878,A -85,B 0,C 180,E1 24481.677,E2 24481.677} C_VEL
LIN {X 0,Y 512.634,Z 401.871,A -85,B 0,C 180,E1 24478.212,E2 24478.212} C_VEL
LIN {X 0,Y 512.639,Z 401.874,A -85,B 0,C 180,E1 24474.628,E2 24474.628} C_VEL
LIN {X 0,Y 512.637,Z 401.877,A -85,B 0,C 180,E1 24471.137,E2 24471.137} C_VEL
LIN {X 0,Y 512.641,Z 401.871,A -85,B 0,C 180,E1 24467.612,E2 24467.612} C_VEL
LIN {X 0,Y 512.63,Z 401.874,A -85,B 0,C 180,E1 24464.067,E2 24464.067} C_VEL
LIN {X 0,Y 512.641,Z 401.874,A -85,B 0,C 180,E1 24460.636,E2 24460.636} C_VEL
LIN {X 0,Y 512.648,Z 401.881,A -85,B 0,C 180,E1 24457.041,E2 24457.041} C_VEL
LIN {X 0,Y 512.627,Z 401.877,A -85,B 0,C 180,E1 24453.544,E2 24453.544} C_VEL
LIN {X 0,Y 512.652,Z 401.875,A -85,B 0,C 180,E1 24450.047,E2 24450.047} C_VEL
LIN {X 0,Y 512.643,Z 401.88,A -85,B 0,C 180,E1 24446.499,E2 24446.499} C_VEL
LIN {X 0,Y 512.627,Z 401.881,A -85,B 0,C 180,E1 24443.077,E2 24443.077} C_VEL
LIN {X 0,Y 512.643,Z 401.869,A -85,B 0,C 180,E1 24439.524,E2 24439.524} C_VEL
LIN {X 0,Y 512.637,Z 401.848,A -85,B 0,C 180,E1 24436.025,E2 24436.025} C_VEL
LIN {X 0,Y 512.675,Z 402.148,A -85,B 0,C 180,E1 24433.248,E2 24433.248} C_VEL
LIN {X 0,Y 513.948,Z 405.371,A -85,B 0,C 180,E1 24432.825,E2 24432.825} C_VEL
LIN {X 0,Y 523.417,Z 425.954,A -85,B 0,C 180,E1 24430.427,E2 24430.427} C_VEL
LIN {X 0,Y 526.706,Z 433.226,A -85,B 0,C 180,E1 24429.632,E2 24429.632} C_VEL
LIN {X 0,Y 525.911,Z 455.704,A -85,B 0,C 180,E1 24428.161,E2 24428.161} C_VEL
LIN {X 0,Y 528.691,Z 473.366,A -85,B 0,C 180,E1 24427.655,E2 24427.655} C_VEL
LIN {X 0,Y 526.215,Z 674.94,A -85,B 0,C 180,E1 24424.557,E2 24424.557} C_VEL
LIN {X 0,Y 525.039,Z 762.276,A -85,B 0,C 180,E1 24423.197,E2 24423.197} C_VEL
LIN {X 0,Y 524.274,Z 783.715,A -85,B 0,C 180,E1 24422.666,E2 24422.666} C_VEL
LIN {X 0,Y 523.344,Z 805.43,A -85,B 0,C 180,E1 24421.922,E2 24421.922} C_VEL
LIN {X 0,Y 522.321,Z 825.122,A -85,B 0,C 180,E1 24421.059,E2 24421.059} C_VEL
LIN {X 0,Y 521.076,Z 844.718,A -85,B 0,C 180,E1 24419.992,E2 24419.992} C_VEL
LIN {X 0,Y 519.712,Z 865.479,A -85,B 0,C 180,E1 24418.625,E2 24418.625} C_VEL
LIN {X 0,Y 518.442,Z 883.735,A -85,B 0,C 180,E1 24417.2,E2 24417.2} C_VEL
LIN {X 0,Y 517.115,Z 901.685,A -85,B 0,C 180,E1 24415.544,E2 24415.544} C_VEL
LIN {X 0,Y 515.9,Z 918.655,A -85,B 0,C 180,E1 24413.715,E2 24413.715} C_VEL
LIN {X 0,Y 514.847,Z 934.161,A -85,B 0,C 180,E1 24411.775,E2 24411.775} C_VEL
LIN {X 0,Y 513.938,Z 948.619,A -85,B 0,C 180,E1 24409.67,E2 24409.67} C_VEL
LIN {X 0,Y 513.213,Z 961.446,A -85,B 0,C 180,E1 24407.461,E2 24407.461} C_VEL
LIN {X 0,Y 512.674,Z 972.806,A -85,B 0,C 180,E1 24405.151,E2 24405.151} C_VEL
LIN {X 0,Y 512.326,Z 982.25,A -85,B 0,C 180,E1 24402.857,E2 24402.857} C_VEL
LIN {X 0,Y 512.109,Z 989.876,A -85,B 0,C 180,E1 24400.577,E2 24400.577} C_VEL
LIN {X 0,Y 511.988,Z 996.14,A -85,B 0,C 180,E1 24398.198,E2 24398.198} C_VEL
LIN {X 0,Y 511.933,Z 1000.82,A -85,B 0,C 180,E1 24395.831,E2 24395.831} C_VEL
LIN {X 0,Y 511.913,Z 1003.784,A -85,B 0,C 180,E1 24393.474,E2 24393.474} C_VEL
LIN {X 0,Y 511.907,Z 1005.305,A -85,B 0,C 180,E1 24391.01,E2 24391.01} C_VEL
LIN {X 0,Y 511.908,Z 1005.26,A -85,B 0,C 180,E1 24388.771,E2 24388.771} C_VEL
LIN {X 0,Y 511.911,Z 1003.675,A -85,B 0,C 180,E1 24386.419,E2 24386.419} C_VEL
LIN {X 0,Y 511.934,Z 1000.637,A -85,B 0,C 180,E1 24384.061,E2 24384.061} C_VEL
LIN {X 0,Y 511.993,Z 995.896,A -85,B 0,C 180,E1 24381.694,E2 24381.694} C_VEL
LIN {X 0,Y 512.121,Z 989.184,A -85,B 0,C 180,E1 24379.2,E2 24379.2} C_VEL
LIN {X 0,Y 512.36,Z 981.17,A -85,B 0,C 180,E1 24376.851,E2 24376.851} C_VEL
LIN {X 0,Y 512.72,Z 971.792,A -85,B 0,C 180,E1 24374.623,E2 24374.623} C_VEL
LIN {X 0,Y 513.285,Z 960.02,A -85,B 0,C 180,E1 24372.278,E2 24372.278} C_VEL
LIN {X 0,Y 514.019,Z 947.117,A -85,B 0,C 180,E1 24370.102,E2 24370.102} C_VEL
LIN {X 0,Y 514.96,Z 932.497,A -85,B 0,C 180,E1 24367.995,E2 24367.995} C_VEL
LIN {X 0,Y 516.044,Z 916.671,A -85,B 0,C 180,E1 24366.055,E2 24366.055} C_VEL
LIN {X 0,Y 517.264,Z 899.651,A -85,B 0,C 180,E1 24364.258,E2 24364.258} C_VEL
LIN {X 0,Y 518.568,Z 881.628,A -85,B 0,C 180,E1 24362.626,E2 24362.626} C_VEL
LIN {X 0,Y 519.895,Z 863.12,A -85,B 0,C 180,E1 24361.203,E2 24361.203} C_VEL
LIN {X 0,Y 521.131,Z 843.802,A -85,B 0,C 180,E1 24359.953,E2 24359.953} C_VEL
LIN {X 0,Y 522.426,Z 823.106,A -85,B 0,C 180,E1 24358.847,E2 24358.847} C_VEL
LIN {X 0,Y 523.431,Z 803.699,A -85,B 0,C 180,E1 24358.008,E2 24358.008} C_VEL
LIN {X 0,Y 524.333,Z 782.345,A -85,B 0,C 180,E1 24357.295,E2 24357.295} C_VEL
LIN {X 0,Y 525.061,Z 760.87,A -85,B 0,C 180,E1 24356.777,E2 24356.777} C_VEL
LIN {X 0,Y 527.851,Z 546.716,A -85,B 0,C 180,E1 24353.468,E2 24353.468} C_VEL
LIN {X 0,Y 528.495,Z 471.161,A -85,B 0,C 180,E1 24352.303,E2 24352.303} C_VEL
LIN {X 0,Y 525.757,Z 454.355,A -85,B 0,C 180,E1 24351.791,E2 24351.791} C_VEL
LIN {X 0,Y 526.468,Z 432.788,A -85,B 0,C 180,E1 24350.352,E2 24350.352} C_VEL
LIN {X 0,Y 514.2,Z 405.803,A -85,B 0,C 180,E1 24347.308,E2 24347.308} C_VEL
LIN {X 0,Y 512.662,Z 402.128,A -85,B 0,C 180,E1 24346.82,E2 24346.82} C_VEL
LIN {X 0,Y 512.629,Z 401.868,A -85,B 0,C 180,E1 24343.651,E2 24343.651} C_VEL
LIN {X 0,Y 512.65,Z 401.876,A -85,B 0,C 180,E1 24340.139,E2 24340.139} C_VEL
LIN {X 0,Y 512.607,Z 401.88,A -85,B 0,C 180,E1 24336.716,E2 24336.716} C_VEL
LIN {X 0,Y 512.603,Z 401.883,A -85,B 0,C 180,E1 24333.205,E2 24333.205} C_VEL
LIN {X 0,Y 512.653,Z 401.877,A -85,B 0,C 180,E1 24329.791,E2 24329.791} C_VEL
LIN {X 0,Y 512.594,Z 401.876,A -85,B 0,C 180,E1 24326.406,E2 24326.406} C_VEL
LIN {X 0,Y 512.585,Z 401.884,A -85,B 0,C 180,E1 24322.962,E2 24322.962} C_VEL
LIN {X 0,Y 512.637,Z 401.88,A -85,B 0,C 180,E1 24319.613,E2 24319.613} C_VEL
LIN {X 0,Y 512.569,Z 401.884,A -85,B 0,C 180,E1 24316.313,E2 24316.313} C_VEL
LIN {X 0,Y 512.572,Z 401.884,A -85,B 0,C 180,E1 24312.734,E2 24312.734} C_VEL
LIN {X 0,Y 512.634,Z 401.88,A -85,B 0,C 180,E1 24309.429,E2 24309.429} C_VEL
LIN {X 0,Y 512.578,Z 401.883,A -85,B 0,C 180,E1 24306.159,E2 24306.159} C_VEL
LIN {X 0,Y 512.601,Z 401.877,A -85,B 0,C 180,E1 24302.683,E2 24302.683} C_VEL
LIN {X 0,Y 512.638,Z 401.877,A -85,B 0,C 180,E1 24299.329,E2 24299.329} C_VEL
LIN {X 0,Y 512.594,Z 401.876,A -85,B 0,C 180,E1 24295.973,E2 24295.973} C_VEL
LIN {X 0,Y 512.621,Z 401.879,A -85,B 0,C 180,E1 24292.491,E2 24292.491} C_VEL
LIN {X 0,Y 512.645,Z 401.877,A -85,B 0,C 180,E1 24289.094,E2 24289.094} C_VEL
LIN {X 0,Y 512.612,Z 401.88,A -85,B 0,C 180,E1 24285.657,E2 24285.657} C_VEL
LIN {X 0,Y 512.629,Z 401.878,A -85,B 0,C 180,E1 24282.129,E2 24282.129} C_VEL
LIN {X 0,Y 512.644,Z 401.867,A -85,B 0,C 180,E1 24278.729,E2 24278.729} C_VEL
LIN {X 0,Y 512.656,Z 402.098,A -85,B 0,C 180,E1 24275.386,E2 24275.386} C_VEL
LIN {X 0,Y 519.933,Z 419.745,A -85,B 0,C 180,E1 24273.009,E2 24273.009} C_VEL
LIN {X 0,Y 523.303,Z 428.72,A -85,B 0,C 180,E1 24271.902,E2 24271.902} C_VEL
LIN {X 0,Y 522.131,Z 452.967,A -85,B 0,C 180,E1 24269.895,E2 24269.895} C_VEL
LIN {X 0,Y 525.123,Z 470,A -85,B 0,C 180,E1 24269.368,E2 24269.368} C_VEL
LIN {X 0,Y 524.024,Z 547.804,A -85,B 0,C 180,E1 24268.166,E2 24268.166} C_VEL
LIN {X 0,Y 523.104,Z 555.497,A -85,B 0,C 180,E1 24268.11,E2 24268.11} C_VEL
LIN {X 0,Y 517.614,Z 576.018,A -85,B 0,C 180,E1 24268.183,E2 24268.183} C_VEL
LIN {X 0,Y 516.895,Z 582.621,A -85,B 0,C 180,E1 24268.128,E2 24268.128} C_VEL
LIN {X 0,Y 515.004,Z 715.633,A -85,B 0,C 180,E1 24266.049,E2 24266.049} C_VEL
LIN {X 0,Y 514.289,Z 736.601,A -85,B 0,C 180,E1 24265.508,E2 24265.508} C_VEL
LIN {X 0,Y 513.423,Z 755.959,A -85,B 0,C 180,E1 24264.799,E2 24264.799} C_VEL
LIN {X 0,Y 512.352,Z 775.189,A -85,B 0,C 180,E1 24263.887,E2 24263.887} C_VEL
LIN {X 0,Y 511.147,Z 794.189,A -85,B 0,C 180,E1 24262.756,E2 24262.756} C_VEL
LIN {X 0,Y 509.93,Z 811.872,A -85,B 0,C 180,E1 24261.47,E2 24261.47} C_VEL
LIN {X 0,Y 508.617,Z 830.142,A -85,B 0,C 180,E1 24259.875,E2 24259.875} C_VEL
LIN {X 0,Y 507.514,Z 846.296,A -85,B 0,C 180,E1 24258.22,E2 24258.22} C_VEL
LIN {X 0,Y 506.509,Z 861.518,A -85,B 0,C 180,E1 24256.368,E2 24256.368} C_VEL
LIN {X 0,Y 505.672,Z 875.023,A -85,B 0,C 180,E1 24254.419,E2 24254.419} C_VEL
LIN {X 0,Y 505.032,Z 886.823,A -85,B 0,C 180,E1 24252.399,E2 24252.399} C_VEL
LIN {X 0,Y 504.548,Z 897.374,A -85,B 0,C 180,E1 24250.238,E2 24250.238} C_VEL
LIN {X 0,Y 504.212,Z 906.566,A -85,B 0,C 180,E1 24247.928,E2 24247.928} C_VEL
LIN {X 0,Y 504.039,Z 913.673,A -85,B 0,C 180,E1 24245.672,E2 24245.672} C_VEL
LIN {X 0,Y 503.955,Z 918.965,A -85,B 0,C 180,E1 24243.47,E2 24243.47} C_VEL
LIN {X 0,Y 503.92,Z 922.72,A -85,B 0,C 180,E1 24241.185,E2 24241.185} C_VEL
LIN {X 0,Y 503.916,Z 924.833,A -85,B 0,C 180,E1 24238.952,E2 24238.952} C_VEL
LIN {X 0,Y 503.906,Z 925.442,A -85,B 0,C 180,E1 24236.64,E2 24236.64} C_VEL
LIN {X 0,Y 503.911,Z 924.48,A -85,B 0,C 180,E1 24234.372,E2 24234.372} C_VEL
LIN {X 0,Y 503.925,Z 921.734,A -85,B 0,C 180,E1 24232.021,E2 24232.021} C_VEL
LIN {X 0,Y 503.962,Z 917.61,A -85,B 0,C 180,E1 24229.829,E2 24229.829} C_VEL
LIN {X 0,Y 504.075,Z 911.675,A -85,B 0,C 180,E1 24227.545,E2 24227.545} C_VEL
LIN {X 0,Y 504.288,Z 904.52,A -85,B 0,C 180,E1 24225.405,E2 24225.405} C_VEL
LIN {X 0,Y 504.646,Z 895.135,A -85,B 0,C 180,E1 24223.168,E2 24223.168} C_VEL
LIN {X 0,Y 505.16,Z 884.401,A -85,B 0,C 180,E1 24221.066,E2 24221.066} C_VEL
LIN {X 0,Y 505.827,Z 872.422,A -85,B 0,C 180,E1 24219.096,E2 24219.096} C_VEL
LIN {X 0,Y 506.704,Z 858.349,A -85,B 0,C 180,E1 24217.139,E2 24217.139} C_VEL
LIN {X 0,Y 507.714,Z 843.283,A -85,B 0,C 180,E1 24215.365,E2 24215.365} C_VEL
LIN {X 0,Y 508.806,Z 827.35,A -85,B 0,C 180,E1 24213.772,E2 24213.772} C_VEL
LIN {X 0,Y 510.099,Z 809.373,A -85,B 0,C 180,E1 24212.244,E2 24212.244} C_VEL
LIN {X 0,Y 511.351,Z 790.97,A -85,B 0,C 180,E1 24210.95,E2 24210.95} C_VEL
LIN {X 0,Y 512.475,Z 772.363,A -85,B 0,C 180,E1 24209.886,E2 24209.886} C_VEL
LIN {X 0,Y 513.475,Z 753.41,A -85,B 0,C 180,E1 24209.021,E2 24209.021} C_VEL
LIN {X 0,Y 514.343,Z 732.877,A -85,B 0,C 180,E1 24208.309,E2 24208.309} C_VEL
LIN {X 0,Y 514.978,Z 712.492,A -85,B 0,C 180,E1 24207.818,E2 24207.818} C_VEL
LIN {X 0,Y 518.284,Z 473.41,A -85,B 0,C 180,E1 24204.126,E2 24204.126} C_VEL
LIN {X 0,Y 518.021,Z 468.674,A -85,B 0,C 180,E1 24204.026,E2 24204.026} C_VEL
LIN {X 0,Y 514.979,Z 452.042,A -85,B 0,C 180,E1 24203.476,E2 24203.476} C_VEL
LIN {X 0,Y 516.052,Z 431.639,A -85,B 0,C 180,E1 24201.755,E2 24201.755} C_VEL
LIN {X 0,Y 509.044,Z 413.573,A -85,B 0,C 180,E1 24199.473,E2 24199.473} C_VEL
LIN {X 0,Y 504.73,Z 403.159,A -85,B 0,C 180,E1 24198.051,E2 24198.051} C_VEL
LIN {X 0,Y 504.704,Z 402.837,A -85,B 0,C 180,E1 24196.829,E2 24196.829} C_VEL
LIN {X 0,Y 504.704,Z 402.841,A -85,B 0,C 180,E1 24193.304,E2 24193.304} C_VEL
LIN {X 0,Y 504.688,Z 402.868,A -85,B 0,C 180,E1 24189.833,E2 24189.833} C_VEL
LIN {X 0,Y 504.701,Z 402.84,A -85,B 0,C 180,E1 24186.285,E2 24186.285} C_VEL
LIN {X 0,Y 504.703,Z 402.862,A -85,B 0,C 180,E1 24182.764,E2 24182.764} C_VEL
LIN {X 0,Y 504.694,Z 402.857,A -85,B 0,C 180,E1 24179.259,E2 24179.259} C_VEL
LIN {X 0,Y 504.695,Z 402.86,A -85,B 0,C 180,E1 24175.703,E2 24175.703} C_VEL
LIN {X 0,Y 504.7,Z 402.868,A -85,B 0,C 180,E1 24172.229,E2 24172.229} C_VEL
LIN {X 0,Y 504.711,Z 402.862,A -85,B 0,C 180,E1 24168.662,E2 24168.662} C_VEL
LIN {X 0,Y 504.692,Z 402.867,A -85,B 0,C 180,E1 24165.146,E2 24165.146} C_VEL
LIN {X 0,Y 504.704,Z 402.857,A -85,B 0,C 180,E1 24161.58,E2 24161.58} C_VEL
LIN {X 0,Y 504.703,Z 402.862,A -85,B 0,C 180,E1 24158.034,E2 24158.034} C_VEL
LIN {X 0,Y 504.695,Z 402.865,A -85,B 0,C 180,E1 24154.497,E2 24154.497} C_VEL
LIN {X 0,Y 504.703,Z 402.858,A -85,B 0,C 180,E1 24150.927,E2 24150.927} C_VEL
LIN {X 0,Y 504.696,Z 402.865,A -85,B 0,C 180,E1 24147.433,E2 24147.433} C_VEL
LIN {X 0,Y 504.702,Z 402.861,A -85,B 0,C 180,E1 24143.962,E2 24143.962} C_VEL
LIN {X 0,Y 504.697,Z 402.855,A -85,B 0,C 180,E1 24140.407,E2 24140.407} C_VEL
LIN {X 0,Y 504.698,Z 402.868,A -85,B 0,C 180,E1 24136.886,E2 24136.886} C_VEL
LIN {X 0,Y 504.702,Z 402.857,A -85,B 0,C 180,E1 24133.286,E2 24133.286} C_VEL
LIN {X 0,Y 504.695,Z 402.857,A -85,B 0,C 180,E1 24129.81,E2 24129.81} C_VEL
LIN {X 0,Y 504.706,Z 402.868,A -85,B 0,C 180,E1 24126.256,E2 24126.256} C_VEL
LIN {X 0,Y 504.693,Z 402.852,A -85,B 0,C 180,E1 24122.726,E2 24122.726} C_VEL
LIN {X 0,Y 504.7,Z 402.858,A -85,B 0,C 180,E1 24119.206,E2 24119.206} C_VEL
LIN {X 0,Y 504.701,Z 402.869,A -85,B 0,C 180,E1 24115.569,E2 24115.569} C_VEL
LIN {X 0,Y 504.689,Z 402.855,A -85,B 0,C 180,E1 24112.129,E2 24112.129} C_VEL
LIN {X 0,Y 504.704,Z 402.857,A -85,B 0,C 180,E1 24108.574,E2 24108.574} C_VEL
LIN {X 0,Y 504.702,Z 402.865,A -85,B 0,C 180,E1 24105.076,E2 24105.076} C_VEL
LIN {X 0,Y 504.698,Z 402.867,A -85,B 0,C 180,E1 24101.52,E2 24101.52} C_VEL
LIN {X 0,Y 504.696,Z 402.861,A -85,B 0,C 180,E1 24097.998,E2 24097.998} C_VEL
LIN {X 0,Y 504.702,Z 402.863,A -85,B 0,C 180,E1 24094.539,E2 24094.539} C_VEL
LIN {X 0,Y 504.706,Z 402.861,A -85,B 0,C 180,E1 24090.964,E2 24090.964} C_VEL
LIN {X 0,Y 504.687,Z 402.862,A -85,B 0,C 180,E1 24087.394,E2 24087.394} C_VEL
LIN {X 0,Y 504.705,Z 402.866,A -85,B 0,C 180,E1 24083.93,E2 24083.93} C_VEL
LIN {X 0,Y 504.706,Z 402.865,A -85,B 0,C 180,E1 24080.365,E2 24080.365} C_VEL
LIN {X 0,Y 504.684,Z 402.846,A -85,B 0,C 180,E1 24076.883,E2 24076.883} C_VEL
LIN {X 0,Y 504.74,Z 403.129,A -85,B 0,C 180,E1 24073.967,E2 24073.967} C_VEL
LIN {X 0,Y 506.047,Z 406.397,A -85,B 0,C 180,E1 24073.521,E2 24073.521} C_VEL
LIN {X 0,Y 514.695,Z 425.121,A -85,B 0,C 180,E1 24071.254,E2 24071.254} C_VEL
LIN {X 0,Y 519.899,Z 436.537,A -85,B 0,C 180,E1 24069.968,E2 24069.968} C_VEL
LIN {X 0,Y 519.174,Z 455.666,A -85,B 0,C 180,E1 24068.698,E2 24068.698} C_VEL
LIN {X 0,Y 522.144,Z 474.7,A -85,B 0,C 180,E1 24068.142,E2 24068.142} C_VEL
LIN {X 0,Y 519.38,Z 693.134,A -85,B 0,C 180,E1 24064.778,E2 24064.778} C_VEL
LIN {X 0,Y 518.333,Z 762.657,A -85,B 0,C 180,E1 24063.675,E2 24063.675} C_VEL
LIN {X 0,Y 517.511,Z 783.973,A -85,B 0,C 180,E1 24063.139,E2 24063.139} C_VEL
LIN {X 0,Y 516.462,Z 806.167,A -85,B 0,C 180,E1 24062.366,E2 24062.366} C_VEL
LIN {X 0,Y 515.318,Z 826.35,A -85,B 0,C 180,E1 24061.464,E2 24061.464} C_VEL
LIN {X 0,Y 513.905,Z 846.724,A -85,B 0,C 180,E1 24060.325,E2 24060.325} C_VEL
LIN {X 0,Y 512.482,Z 866.287,A -85,B 0,C 180,E1 24059.003,E2 24059.003} C_VEL
LIN {X 0,Y 511.087,Z 884.407,A -85,B 0,C 180,E1 24057.562,E2 24057.562} C_VEL
LIN {X 0,Y 509.652,Z 902.29,A -85,B 0,C 180,E1 24055.883,E2 24055.883} C_VEL
LIN {X 0,Y 508.388,Z 918.224,A -85,B 0,C 180,E1 24054.139,E2 24054.139} C_VEL
LIN {X 0,Y 507.247,Z 933.312,A -85,B 0,C 180,E1 24052.24,E2 24052.24} C_VEL
LIN {X 0,Y 506.226,Z 947.854,A -85,B 0,C 180,E1 24050.103,E2 24050.103} C_VEL
LIN {X 0,Y 505.424,Z 960.528,A -85,B 0,C 180,E1 24047.911,E2 24047.911} C_VEL
LIN {X 0,Y 504.796,Z 972.29,A -85,B 0,C 180,E1 24045.511,E2 24045.511} C_VEL
LIN {X 0,Y 504.393,Z 981.843,A -85,B 0,C 180,E1 24043.179,E2 24043.179} C_VEL
LIN {X 0,Y 504.138,Z 989.522,A -85,B 0,C 180,E1 24040.862,E2 24040.862} C_VEL
LIN {X 0,Y 503.998,Z 996.14,A -85,B 0,C 180,E1 24038.329,E2 24038.329} C_VEL
LIN {X 0,Y 503.935,Z 1000.82,A -85,B 0,C 180,E1 24035.924,E2 24035.924} C_VEL
LIN {X 0,Y 503.913,Z 1003.785,A -85,B 0,C 180,E1 24033.529,E2 24033.529} C_VEL
LIN {X 0,Y 503.907,Z 1005.304,A -85,B 0,C 180,E1 24031.026,E2 24031.026} C_VEL
LIN {X 0,Y 503.908,Z 1005.26,A -85,B 0,C 180,E1 24028.752,E2 24028.752} C_VEL
LIN {X 0,Y 503.911,Z 1003.675,A -85,B 0,C 180,E1 24026.362,E2 24026.362} C_VEL
LIN {X 0,Y 503.937,Z 1000.637,A -85,B 0,C 180,E1 24023.966,E2 24023.966} C_VEL
LIN {X 0,Y 504.001,Z 995.896,A -85,B 0,C 180,E1 24021.561,E2 24021.561} C_VEL
LIN {X 0,Y 504.146,Z 989.181,A -85,B 0,C 180,E1 24019.026,E2 24019.026} C_VEL
LIN {X 0,Y 504.407,Z 981.439,A -85,B 0,C 180,E1 24016.709,E2 24016.709} C_VEL
LIN {X 0,Y 504.822,Z 971.793,A -85,B 0,C 180,E1 24014.377,E2 24014.377} C_VEL
LIN {X 0,Y 505.443,Z 960.203,A -85,B 0,C 180,E1 24012.028,E2 24012.028} C_VEL
LIN {X 0,Y 506.224,Z 947.886,A -85,B 0,C 180,E1 24009.902,E2 24009.902} C_VEL
LIN {X 0,Y 507.244,Z 933.348,A -85,B 0,C 180,E1 24007.765,E2 24007.765} C_VEL
LIN {X 0,Y 508.391,Z 918.191,A -85,B 0,C 180,E1 24005.857,E2 24005.857} C_VEL
LIN {X 0,Y 509.744,Z 901.127,A -85,B 0,C 180,E1 24004.002,E2 24004.002} C_VEL
LIN {X 0,Y 511.137,Z 883.794,A -85,B 0,C 180,E1 24002.384,E2 24002.384} C_VEL
LIN {X 0,Y 512.575,Z 865.162,A -85,B 0,C 180,E1 24000.914,E2 24000.914} C_VEL
LIN {X 0,Y 514.028,Z 844.804,A -85,B 0,C 180,E1 23999.559,E2 23999.559} C_VEL
LIN {X 0,Y 515.389,Z 825.234,A -85,B 0,C 180,E1 23998.482,E2 23998.482} C_VEL
LIN {X 0,Y 516.533,Z 804.825,A -85,B 0,C 180,E1 23997.579,E2 23997.579} C_VEL
LIN {X 0,Y 517.56,Z 782.905,A -85,B 0,C 180,E1 23996.83,E2 23996.83} C_VEL
LIN {X 0,Y 518.355,Z 761.62,A -85,B 0,C 180,E1 23996.305,E2 23996.305} C_VEL
LIN {X 0,Y 520.019,Z 643.588,A -85,B 0,C 180,E1 23994.46,E2 23994.46} C_VEL
LIN {X 0,Y 521.958,Z 472.929,A -85,B 0,C 180,E1 23991.836,E2 23991.836} C_VEL
LIN {X 0,Y 518.968,Z 454.695,A -85,B 0,C 180,E1 23991.286,E2 23991.286} C_VEL
LIN {X 0,Y 519.723,Z 436.387,A -85,B 0,C 180,E1 23990.053,E2 23990.053} C_VEL
LIN {X 0,Y 507.943,Z 410.484,A -85,B 0,C 180,E1 23987.076,E2 23987.076} C_VEL
LIN {X 0,Y 504.77,Z 403.269,A -85,B 0,C 180,E1 23986.162,E2 23986.162} C_VEL
LIN {X 0,Y 504.675,Z 402.86,A -85,B 0,C 180,E1 23985.336,E2 23985.336} C_VEL
LIN {X 0,Y 504.704,Z 402.86,A -85,B 0,C 180,E1 23981.856,E2 23981.856} C_VEL
LIN {X 0,Y 504.703,Z 402.865,A -85,B 0,C 180,E1 23978.322,E2 23978.322} C_VEL
LIN {X 0,Y 504.659,Z 402.87,A -85,B 0,C 180,E1 23974.898,E2 23974.898} C_VEL
LIN {X 0,Y 504.673,Z 402.871,A -85,B 0,C 180,E1 23971.37,E2 23971.37} C_VEL
LIN {X 0,Y 504.698,Z 402.868,A -85,B 0,C 180,E1 23968.003,E2 23968.003} C_VEL
LIN {X 0,Y 504.643,Z 402.871,A -85,B 0,C 180,E1 23964.584,E2 23964.584} C_VEL
LIN {X 0,Y 504.655,Z 402.868,A -85,B 0,C 180,E1 23961.136,E2 23961.136} C_VEL
LIN {X 0,Y 504.679,Z 402.866,A -85,B 0,C 180,E1 23957.764,E2 23957.764} C_VEL
LIN {X 0,Y 504.623,Z 402.868,A -85,B 0,C 180,E1 23954.457,E2 23954.457} C_VEL
LIN {X 0,Y 504.665,Z 402.87,A -85,B 0,C 180,E1 23951.08,E2 23951.08} C_VEL
LIN {X 0,Y 504.662,Z 402.866,A -85,B 0,C 180,E1 23947.742,E2 23947.742} C_VEL
LIN {X 0,Y 504.642,Z 402.87,A -85,B 0,C 180,E1 23944.318,E2 23944.318} C_VEL
LIN {X 0,Y 504.691,Z 402.869,A -85,B 0,C 180,E1 23940.908,E2 23940.908} C_VEL
LIN {X 0,Y 504.67,Z 402.872,A -85,B 0,C 180,E1 23937.615,E2 23937.615} C_VEL
LIN {X 0,Y 504.659,Z 402.869,A -85,B 0,C 180,E1 23934.086,E2 23934.086} C_VEL
LIN {X 0,Y 504.701,Z 402.867,A -85,B 0,C 180,E1 23930.651,E2 23930.651} C_VEL
LIN {X 0,Y 504.7,Z 402.87,A -85,B 0,C 180,E1 23927.18,E2 23927.18} C_VEL
LIN {X 0,Y 504.674,Z 402.869,A -85,B 0,C 180,E1 23923.778,E2 23923.778} C_VEL
LIN {X 0,Y 504.705,Z 402.866,A -85,B 0,C 180,E1 23920.319,E2 23920.319} C_VEL
LIN {X 0,Y 504.707,Z 402.867,A -85,B 0,C 180,E1 23916.782,E2 23916.782} C_VEL
LIN {X 0,Y 504.743,Z 403.158,A -85,B 0,C 180,E1 23916.071,E2 23916.071} C_VEL
LIN {X 0,Y 512.259,Z 421.211,A -85,B 0,C 180,E1 23913.575,E2 23913.575} C_VEL
LIN {X 0,Y 516.452,Z 432.175,A -85,B 0,C 180,E1 23912.187,E2 23912.187} C_VEL
LIN {X 0,Y 515.329,Z 452.946,A -85,B 0,C 180,E1 23910.45,E2 23910.45} C_VEL
LIN {X 0,Y 518.606,Z 471.167,A -85,B 0,C 180,E1 23909.865,E2 23909.865} C_VEL
LIN {X 0,Y 516.895,Z 582.621,A -85,B 0,C 180,E1 23908.128,E2 23908.128} C_VEL
LIN {X 0,Y 515.963,Z 590.314,A -85,B 0,C 180,E1 23908.072,E2 23908.072} C_VEL
LIN {X 0,Y 510.476,Z 610.833,A -85,B 0,C 180,E1 23908.145,E2 23908.145} C_VEL
LIN {X 0,Y 509.75,Z 617.433,A -85,B 0,C 180,E1 23908.089,E2 23908.089} C_VEL
LIN {X 0,Y 508.16,Z 716.387,A -85,B 0,C 180,E1 23906.505,E2 23906.505} C_VEL
LIN {X 0,Y 507.396,Z 737.391,A -85,B 0,C 180,E1 23905.954,E2 23905.954} C_VEL
LIN {X 0,Y 506.473,Z 756.525,A -85,B 0,C 180,E1 23905.243,E2 23905.243} C_VEL
LIN {X 0,Y 505.341,Z 775.421,A -85,B 0,C 180,E1 23904.339,E2 23904.339} C_VEL
LIN {X 0,Y 504.048,Z 794.45,A -85,B 0,C 180,E1 23903.197,E2 23903.197} C_VEL
LIN {X 0,Y 502.763,Z 811.676,A -85,B 0,C 180,E1 23901.938,E2 23901.938} C_VEL
LIN {X 0,Y 501.374,Z 828.99,A -85,B 0,C 180,E1 23900.417,E2 23900.417} C_VEL
LIN {X 0,Y 500.041,Z 845.172,A -85,B 0,C 180,E1 23898.711,E2 23898.711} C_VEL
LIN {X 0,Y 498.711,Z 862.637,A -85,B 0,C 180,E1 23896.527,E2 23896.527} C_VEL
LIN {X 0,Y 497.796,Z 876.302,A -85,B 0,C 180,E1 23894.501,E2 23894.501} C_VEL
LIN {X 0,Y 497.082,Z 888.38,A -85,B 0,C 180,E1 23892.359,E2 23892.359} C_VEL
LIN {X 0,Y 496.574,Z 898.512,A -85,B 0,C 180,E1 23890.193,E2 23890.193} C_VEL
LIN {X 0,Y 496.238,Z 906.872,A -85,B 0,C 180,E1 23888.018,E2 23888.018} C_VEL
LIN {X 0,Y 496.046,Z 914.027,A -85,B 0,C 180,E1 23885.677,E2 23885.677} C_VEL
LIN {X 0,Y 495.955,Z 919.312,A -85,B 0,C 180,E1 23883.389,E2 23883.389} C_VEL
LIN {X 0,Y 495.924,Z 923.152,A -85,B 0,C 180,E1 23880.935,E2 23880.935} C_VEL
LIN {X 0,Y 495.908,Z 925.015,A -85,B 0,C 180,E1 23878.672,E2 23878.672} C_VEL
LIN {X 0,Y 495.905,Z 925.382,A -85,B 0,C 180,E1 23876.328,E2 23876.328} C_VEL
LIN {X 0,Y 495.912,Z 924.197,A -85,B 0,C 180,E1 23874.028,E2 23874.028} C_VEL
LIN {X 0,Y 495.92,Z 921.501,A -85,B 0,C 180,E1 23871.772,E2 23871.772} C_VEL
LIN {X 0,Y 495.973,Z 917.248,A -85,B 0,C 180,E1 23869.548,E2 23869.548} C_VEL
LIN {X 0,Y 496.114,Z 911.085,A -85,B 0,C 180,E1 23867.197,E2 23867.197} C_VEL
LIN {X 0,Y 496.364,Z 903.434,A -85,B 0,C 180,E1 23864.939,E2 23864.939} C_VEL
LIN {X 0,Y 496.764,Z 894.44,A -85,B 0,C 180,E1 23862.788,E2 23862.788} C_VEL
LIN {X 0,Y 497.392,Z 882.945,A -85,B 0,C 180,E1 23860.538,E2 23860.538} C_VEL
LIN {X 0,Y 498.212,Z 869.925,A -85,B 0,C 180,E1 23858.422,E2 23858.422} C_VEL
LIN {X 0,Y 499.17,Z 856.088,A -85,B 0,C 180,E1 23856.529,E2 23856.529} C_VEL
LIN {X 0,Y 500.386,Z 840.576,A -85,B 0,C 180,E1 23854.697,E2 23854.697} C_VEL
LIN {X 0,Y 501.699,Z 824.392,A -85,B 0,C 180,E1 23853.082,E2 23853.082} C_VEL
LIN {X 0,Y 503.029,Z 807.289,A -85,B 0,C 180,E1 23851.649,E2 23851.649} C_VEL
LIN {X 0,Y 504.297,Z 790.205,A -85,B 0,C 180,E1 23850.452,E2 23850.452} C_VEL
LIN {X 0,Y 505.531,Z 771.315,A -85,B 0,C 180,E1 23849.374,E2 23849.374} C_VEL
LIN {X 0,Y 506.594,Z 751.9,A -85,B 0,C 180,E1 23848.499,E2 23848.499} C_VEL
LIN {X 0,Y 507.496,Z 731.862,A -85,B 0,C 180,E1 23847.817,E2 23847.817} C_VEL
LIN {X 0,Y 508.144,Z 710.879,A -85,B 0,C 180,E1 23847.323,E2 23847.323} C_VEL
LIN {X 0,Y 511.737,Z 473.814,A -85,B 0,C 180,E1 23843.616,E2 23843.616} C_VEL
LIN {X 0,Y 511.306,Z 469.159,A -85,B 0,C 180,E1 23843.501,E2 23843.501} C_VEL
LIN {X 0,Y 508.171,Z 452.261,A -85,B 0,C 180,E1 23842.934,E2 23842.934} C_VEL
LIN {X 0,Y 509.006,Z 434.581,A -85,B 0,C 180,E1 23841.412,E2 23841.412} C_VEL
LIN {X 0,Y 501.922,Z 416.604,A -85,B 0,C 180,E1 23839.089,E2 23839.089} C_VEL
LIN {X 0,Y 496.795,Z 404.068,A -85,B 0,C 180,E1 23837.34,E2 23837.34} C_VEL
LIN {X 0,Y 496.747,Z 403.839,A -85,B 0,C 180,E1 23833.871,E2 23833.871} C_VEL
LIN {X 0,Y 496.757,Z 403.86,A -85,B 0,C 180,E1 23830.234,E2 23830.234} C_VEL
LIN {X 0,Y 496.759,Z 403.821,A -85,B 0,C 180,E1 23826.763,E2 23826.763} C_VEL
LIN {X 0,Y 496.763,Z 403.852,A -85,B 0,C 180,E1 23823.2,E2 23823.2} C_VEL
LIN {X 0,Y 496.751,Z 403.849,A -85,B 0,C 180,E1 23819.653,E2 23819.653} C_VEL
LIN {X 0,Y 496.766,Z 403.853,A -85,B 0,C 180,E1 23816.113,E2 23816.113} C_VEL
LIN {X 0,Y 496.763,Z 403.854,A -85,B 0,C 180,E1 23812.47,E2 23812.47} C_VEL
LIN {X 0,Y 496.756,Z 403.854,A -85,B 0,C 180,E1 23808.99,E2 23808.99} C_VEL
LIN {X 0,Y 496.759,Z 403.853,A -85,B 0,C 180,E1 23805.374,E2 23805.374} C_VEL
LIN {X 0,Y 496.759,Z 403.846,A -85,B 0,C 180,E1 23801.863,E2 23801.863} C_VEL
LIN {X 0,Y 496.767,Z 403.85,A -85,B 0,C 180,E1 23798.281,E2 23798.281} C_VEL
LIN {X 0,Y 496.753,Z 403.856,A -85,B 0,C 180,E1 23794.724,E2 23794.724} C_VEL
LIN {X 0,Y 496.765,Z 403.844,A -85,B 0,C 180,E1 23791.15,E2 23791.15} C_VEL
LIN {X 0,Y 496.759,Z 403.853,A -85,B 0,C 180,E1 23787.577,E2 23787.577} C_VEL
LIN {X 0,Y 496.762,Z 403.85,A -85,B 0,C 180,E1 23783.99,E2 23783.99} C_VEL
LIN {X 0,Y 496.757,Z 403.843,A -85,B 0,C 180,E1 23780.378,E2 23780.378} C_VEL
LIN {X 0,Y 496.76,Z 403.857,A -85,B 0,C 180,E1 23776.849,E2 23776.849} C_VEL
LIN {X 0,Y 496.763,Z 403.846,A -85,B 0,C 180,E1 23773.265,E2 23773.265} C_VEL
LIN {X 0,Y 496.757,Z 403.844,A -85,B 0,C 180,E1 23769.734,E2 23769.734} C_VEL
LIN {X 0,Y 496.768,Z 403.858,A -85,B 0,C 180,E1 23766.121,E2 23766.121} C_VEL
LIN {X 0,Y 496.753,Z 403.841,A -85,B 0,C 180,E1 23762.538,E2 23762.538} C_VEL
LIN {X 0,Y 496.767,Z 403.845,A -85,B 0,C 180,E1 23758.962,E2 23758.962} C_VEL
LIN {X 0,Y 496.759,Z 403.856,A -85,B 0,C 180,E1 23755.382,E2 23755.382} C_VEL
LIN {X 0,Y 496.757,Z 403.845,A -85,B 0,C 180,E1 23751.901,E2 23751.901} C_VEL
LIN {X 0,Y 496.755,Z 403.848,A -85,B 0,C 180,E1 23748.271,E2 23748.271} C_VEL
LIN {X 0,Y 496.764,Z 403.85,A -85,B 0,C 180,E1 23744.712,E2 23744.712} C_VEL
LIN {X 0,Y 496.766,Z 403.857,A -85,B 0,C 180,E1 23741.084,E2 23741.084} C_VEL
LIN {X 0,Y 496.755,Z 403.854,A -85,B 0,C 180,E1 23737.5,E2 23737.5} C_VEL
LIN {X 0,Y 496.757,Z 403.852,A -85,B 0,C 180,E1 23733.846,E2 23733.846} C_VEL
LIN {X 0,Y 496.763,Z 403.856,A -85,B 0,C 180,E1 23730.322,E2 23730.322} C_VEL
LIN {X 0,Y 496.765,Z 403.856,A -85,B 0,C 180,E1 23726.807,E2 23726.807} C_VEL
LIN {X 0,Y 496.749,Z 403.858,A -85,B 0,C 180,E1 23723.237,E2 23723.237} C_VEL
LIN {X 0,Y 496.773,Z 403.846,A -85,B 0,C 180,E1 23719.715,E2 23719.715} C_VEL
LIN {X 0,Y 496.76,Z 403.821,A -85,B 0,C 180,E1 23716.103,E2 23716.103} C_VEL
LIN {X 0,Y 496.79,Z 404.127,A -85,B 0,C 180,E1 23714.703,E2 23714.703} C_VEL
LIN {X 0,Y 498.167,Z 407.491,A -85,B 0,C 180,E1 23714.232,E2 23714.232} C_VEL
LIN {X 0,Y 506.385,Z 425.165,A -85,B 0,C 180,E1 23712.019,E2 23712.019} C_VEL
LIN {X 0,Y 513.127,Z 440.115,A -85,B 0,C 180,E1 23710.292,E2 23710.292} C_VEL
LIN {X 0,Y 512.491,Z 455.692,A -85,B 0,C 180,E1 23709.248,E2 23709.248} C_VEL
LIN {X 0,Y 515.633,Z 476.214,A -85,B 0,C 180,E1 23708.639,E2 23708.639} C_VEL
LIN {X 0,Y 512.628,Z 696.18,A -85,B 0,C 180,E1 23705.218,E2 23705.218} C_VEL
LIN {X 0,Y 511.645,Z 762.724,A -85,B 0,C 180,E1 23704.167,E2 23704.167} C_VEL
LIN {X 0,Y 510.829,Z 783.281,A -85,B 0,C 180,E1 23703.652,E2 23703.652} C_VEL
LIN {X 0,Y 509.698,Z 805.349,A -85,B 0,C 180,E1 23702.886,E2 23702.886} C_VEL
LIN {X 0,Y 508.502,Z 825.128,A -85,B 0,C 180,E1 23702.001,E2 23702.001} C_VEL
LIN {X 0,Y 507.032,Z 844.711,A -85,B 0,C 180,E1 23700.912,E2 23700.912} C_VEL
LIN {X 0,Y 505.462,Z 864.911,A -85,B 0,C 180,E1 23699.555,E2 23699.555} C_VEL
LIN {X 0,Y 503.873,Z 883.733,A -85,B 0,C 180,E1 23698.055,E2 23698.055} C_VEL
LIN {X 0,Y 502.313,Z 901.682,A -85,B 0,C 180,E1 23696.354,E2 23696.354} C_VEL
LIN {X 0,Y 500.873,Z 918.147,A -85,B 0,C 180,E1 23694.535,E2 23694.535} C_VEL
LIN {X 0,Y 499.612,Z 933.313,A -85,B 0,C 180,E1 23692.599,E2 23692.599} C_VEL
LIN {X 0,Y 498.489,Z 947.852,A -85,B 0,C 180,E1 23690.428,E2 23690.428} C_VEL
LIN {X 0,Y 497.621,Z 960.174,A -85,B 0,C 180,E1 23688.269,E2 23688.269} C_VEL
LIN {X 0,Y 496.932,Z 971.773,A -85,B 0,C 180,E1 23685.883,E2 23685.883} C_VEL
LIN {X 0,Y 496.469,Z 981.422,A -85,B 0,C 180,E1 23683.512,E2 23683.512} C_VEL
LIN {X 0,Y 496.165,Z 989.522,A -85,B 0,C 180,E1 23681.039,E2 23681.039} C_VEL
LIN {X 0,Y 496.007,Z 996.141,A -85,B 0,C 180,E1 23678.464,E2 23678.464} C_VEL
LIN {X 0,Y 495.937,Z 1000.82,A -85,B 0,C 180,E1 23676.02,E2 23676.02} C_VEL
LIN {X 0,Y 495.912,Z 1003.785,A -85,B 0,C 180,E1 23673.586,E2 23673.586} C_VEL
LIN {X 0,Y 495.908,Z 1005.304,A -85,B 0,C 180,E1 23671.042,E2 23671.042} C_VEL
LIN {X 0,Y 495.908,Z 1005.259,A -85,B 0,C 180,E1 23668.732,E2 23668.732} C_VEL
LIN {X 0,Y 495.91,Z 1003.674,A -85,B 0,C 180,E1 23666.303,E2 23666.303} C_VEL
LIN {X 0,Y 495.939,Z 1000.637,A -85,B 0,C 180,E1 23663.869,E2 23663.869} C_VEL
LIN {X 0,Y 496.009,Z 995.896,A -85,B 0,C 180,E1 23661.424,E2 23661.424} C_VEL
LIN {X 0,Y 496.173,Z 989.183,A -85,B 0,C 180,E1 23658.848,E2 23658.848} C_VEL
LIN {X 0,Y 496.468,Z 981.438,A -85,B 0,C 180,E1 23656.493,E2 23656.493} C_VEL
LIN {X 0,Y 496.935,Z 971.71,A -85,B 0,C 180,E1 23654.103,E2 23654.103} C_VEL
LIN {X 0,Y 497.62,Z 960.201,A -85,B 0,C 180,E1 23651.736,E2 23651.736} C_VEL
LIN {X 0,Y 498.523,Z 947.348,A -85,B 0,C 180,E1 23649.493,E2 23649.493} C_VEL
LIN {X 0,Y 499.609,Z 933.349,A -85,B 0,C 180,E1 23647.406,E2 23647.406} C_VEL
LIN {X 0,Y 500.869,Z 918.19,A -85,B 0,C 180,E1 23645.47,E2 23645.47} C_VEL
LIN {X 0,Y 502.358,Z 901.129,A -85,B 0,C 180,E1 23643.591,E2 23643.591} C_VEL
LIN {X 0,Y 503.929,Z 883.086,A -85,B 0,C 180,E1 23641.89,E2 23641.89} C_VEL
LIN {X 0,Y 505.463,Z 864.911,A -85,B 0,C 180,E1 23640.445,E2 23640.445} C_VEL
LIN {X 0,Y 507.025,Z 844.8,A -85,B 0,C 180,E1 23639.093,E2 23639.093} C_VEL
LIN {X 0,Y 508.496,Z 825.237,A -85,B 0,C 180,E1 23638.004,E2 23638.004} C_VEL
LIN {X 0,Y 509.732,Z 804.789,A -85,B 0,C 180,E1 23637.091,E2 23637.091} C_VEL
LIN {X 0,Y 510.842,Z 783.047,A -85,B 0,C 180,E1 23636.341,E2 23636.341} C_VEL
LIN {X 0,Y 511.647,Z 762.589,A -85,B 0,C 180,E1 23635.83,E2 23635.83} C_VEL
LIN {X 0,Y 512.717,Z 686.891,A -85,B 0,C 180,E1 23634.645,E2 23634.645} C_VEL
LIN {X 0,Y 515.492,Z 474.928,A -85,B 0,C 180,E1 23631.364,E2 23631.364} C_VEL
LIN {X 0,Y 512.23,Z 454.577,A -85,B 0,C 180,E1 23630.738,E2 23630.738} C_VEL
LIN {X 0,Y 512.946,Z 440.085,A -85,B 0,C 180,E1 23629.749,E2 23629.749} C_VEL
LIN {X 0,Y 502.082,Z 415.757,A -85,B 0,C 180,E1 23626.922,E2 23626.922} C_VEL
LIN {X 0,Y 496.811,Z 404.312,A -85,B 0,C 180,E1 23625.434,E2 23625.434} C_VEL
LIN {X 0,Y 496.742,Z 403.854,A -85,B 0,C 180,E1 23624.891,E2 23624.891} C_VEL
LIN {X 0,Y 496.734,Z 403.862,A -85,B 0,C 180,E1 23621.316,E2 23621.316} C_VEL
LIN {X 0,Y 496.771,Z 403.855,A -85,B 0,C 180,E1 23617.87,E2 23617.87} C_VEL
LIN {X 0,Y 496.751,Z 403.855,A -85,B 0,C 180,E1 23614.304,E2 23614.304} C_VEL
LIN {X 0,Y 496.714,Z 403.861,A -85,B 0,C 180,E1 23610.884,E2 23610.884} C_VEL
LIN {X 0,Y 496.739,Z 403.856,A -85,B 0,C 180,E1 23607.428,E2 23607.428} C_VEL
LIN {X 0,Y 496.741,Z 403.856,A -85,B 0,C 180,E1 23603.991,E2 23603.991} C_VEL
LIN {X 0,Y 496.695,Z 403.857,A -85,B 0,C 180,E1 23600.613,E2 23600.613} C_VEL
LIN {X 0,Y 496.725,Z 403.86,A -85,B 0,C 180,E1 23597.211,E2 23597.211} C_VEL
LIN {X 0,Y 496.714,Z 403.857,A -85,B 0,C 180,E1 23593.859,E2 23593.859} C_VEL
LIN {X 0,Y 496.69,Z 403.862,A -85,B 0,C 180,E1 23590.438,E2 23590.438} C_VEL
LIN {X 0,Y 496.741,Z 403.86,A -85,B 0,C 180,E1 23587.052,E2 23587.052} C_VEL
LIN {X 0,Y 496.736,Z 403.861,A -85,B 0,C 180,E1 23583.577,E2 23583.577} C_VEL
